Staubli VAL3: Cercle10.pjx

--- Cercle10.pjx ---
Parameters version=s7.3.1 stackSize=5000 millimeterUnit=true
Program file=start.pgx
Program file=stop.pgx
Data file=Cercle10.dtx

--- Cercle10.dtx ---
public frame fReference = {x=1500, y=200, z=-689.53, rz=90, fatherId=world[0]}
public jointRx jPark = {j3=90, j5=90}
public jointRx jJoint = {j1=-0.42016, j2=47.67737, j3=89.12207, j5=43.20056, j6=178.21616}
public mdesc mNomSpeed = {blend=off}
public mdesc mSpeed[30]
  [0] = {tmax=30, rmax=100, leave=0.1, reach=0.1, blend=cartesian}
  [1] = {tmax=30, rmax=100, leave=0.1, reach=0.1, blend=cartesian}
  [2] = {tmax=30, rmax=100, leave=0.1, reach=0.1, blend=cartesian}
  [3] = {tmax=30, rmax=100, leave=0.1, reach=0.1, blend=cartesian}
  [4] = {tmax=30, rmax=100, leave=0.1, reach=0.1, blend=cartesian}
  [5] = {tmax=30, rmax=100, leave=0.1, reach=0.1, blend=cartesian}
  [6] = {tmax=30, rmax=100, leave=0.1, reach=0.1, blend=cartesian}
  [7] = {tmax=30, rmax=100, leave=0.1, reach=0.1, blend=cartesian}
  [8] = {tmax=30, rmax=100, leave=0.1, reach=0.1, blend=cartesian}
  [9] = {tmax=30, rmax=100, leave=0.1, reach=0.1, blend=cartesian}
  [10] = {tmax=30, rmax=100, leave=0.1, reach=0.1, blend=cartesian}
  [11] = {tmax=30, rmax=100, leave=0.1, reach=0.1, blend=cartesian}
  [12] = {tmax=30, rmax=100, leave=0.1, reach=0.1, blend=cartesian}
  [13] = {tmax=30, rmax=100, leave=0.1, reach=0.1, blend=cartesian}
  [14] = {tmax=30, rmax=100, leave=0.1, reach=0.1, blend=cartesian}
  [15] = {tmax=30, rmax=100, leave=0.1, reach=0.1, blend=cartesian}
  [16] = {tmax=30, rmax=100, leave=0.1, reach=0.1, blend=cartesian}
  [17] = {tmax=30, rmax=100, leave=0.1, reach=0.1, blend=cartesian}
  [18] = {tmax=30, rmax=100, leave=0.1, reach=0.1, blend=cartesian}
  [19] = {tmax=30, rmax=100, leave=0.1, reach=0.1, blend=cartesian}
  [20] = {tmax=30, rmax=100, leave=0.1, reach=0.1, blend=cartesian}
  [21] = {tmax=30, rmax=100, leave=0.1, reach=0.1, blend=cartesian}
  [22] = {tmax=30, rmax=100, leave=0.1, reach=0.1, blend=cartesian}
  [23] = {tmax=30, rmax=100, leave=0.1, reach=0.1, blend=cartesian}
  [24] = {tmax=30, rmax=100, leave=0.1, reach=0.1, blend=cartesian}
  [25] = {tmax=30, rmax=100, leave=0.1, reach=0.1, blend=cartesian}
  [26] = {tmax=30, rmax=100, leave=0.1, reach=0.1, blend=cartesian}
  [27] = {tmax=30, rmax=100, leave=0.1, reach=0.1, blend=cartesian}
  [28] = {tmax=30, rmax=100, leave=0.1, reach=0.1, blend=cartesian}
  [29] = {tmax=30, rmax=100, leave=0.1, reach=0.1, blend=cartesian}
public num nTraj
num nTimeStop
num nTimeStart
num nMode
num nEtat
public pointRx pPoint[1370]
  [0] = {x=-211, z=100, rx=-180, rz=88.636, shoulder=lefty, elbow=epositive, wrist=wpositive, fatherId=fReference[0]}
  [1] = {x=-211, rx=-180, rz=88.636, shoulder=lefty, elbow=epositive, wrist=wpositive, fatherId=fReference[0]}
  [2] = {x=-211, rx=-180, rz=88.636, shoulder=lefty, elbow=epositive, wrist=wpositive, fatherId=fReference[0]}
  [3] = {x=-210.761, y=-10.04, rx=-180, rz=85.909, shoulder=lefty, elbow=epositive, wrist=wpositive, fatherId=fReference[0]}
  [4] = {x=-210.045, y=-20.057, rx=-180, rz=83.182, shoulder=lefty, elbow=epositive, wrist=wpositive, fatherId=fReference[0]}
  [5] = {x=-208.852, y=-30.028, rx=-180, rz=80.455, shoulder=lefty, elbow=epositive, wrist=wpositive, fatherId=fReference[0]}
  [6] = {x=-207.187, y=-39.932, rx=-180, rz=77.727, shoulder=lefty, elbow=epositive, wrist=wpositive, fatherId=fReference[0]}
  [7] = {x=-205.052, y=-49.745, rx=-180, rz=75, shoulder=lefty, elbow=epositive, wrist=wpositive, fatherId=fReference[0]}
  [8] = {x=-202.453, y=-59.446, rx=-180, rz=72.273, shoulder=lefty, elbow=epositive, wrist=wpositive, fatherId=fReference[0]}
  [9] = {x=-199.395, y=-69.011, rx=-180, rz=69.545, shoulder=lefty, elbow=epositive, wrist=wpositive, fatherId=fReference[0]}
  [10] = {x=-195.886, y=-78.421, rx=-180, rz=66.818, shoulder=lefty, elbow=epositive, wrist=wpositive, fatherId=fReference[0]}
  [11] = {x=-191.932, y=-87.653, rx=-180, rz=64.091, shoulder=lefty, elbow=epositive, wrist=wpositive, fatherId=fReference[0]}
  [12] = {x=-187.544, y=-96.686, rx=-180, rz=61.364, shoulder=lefty, elbow=epositive, wrist=wpositive, fatherId=fReference[0]}
  [13] = {x=-182.731, y=-105.5, rx=180, rz=58.636, shoulder=lefty, elbow=epositive, wrist=wpositive, fatherId=fReference[0]}
  [14] = {x=-177.505, y=-114.075, rx=-180, rz=55.909, shoulder=lefty, elbow=epositive, wrist=wpositive, fatherId=fReference[0]}
  [15] = {x=-171.876, y=-122.392, rx=-180, rz=53.182, shoulder=lefty, elbow=epositive, wrist=wpositive, fatherId=fReference[0]}
  [16] = {x=-165.857, y=-130.432, rx=-180, rz=50.455, shoulder=lefty, elbow=epositive, wrist=wpositive, fatherId=fReference[0]}
  [17] = {x=-159.463, y=-138.176, rx=-180, rz=47.727, shoulder=lefty, elbow=epositive, wrist=wpositive, fatherId=fReference[0]}
  [18] = {x=-152.708, y=-145.607, rx=-180, rz=45, shoulder=lefty, elbow=epositive, wrist=wpositive, fatherId=fReference[0]}
  [19] = {x=-145.607, y=-152.708, rx=-180, rz=42.273, shoulder=lefty, elbow=epositive, wrist=wpositive, fatherId=fReference[0]}
  [20] = {x=-138.176, y=-159.463, rx=-180, rz=39.545, shoulder=lefty, elbow=epositive, wrist=wpositive, fatherId=fReference[0]}
  [21] = {x=-130.432, y=-165.857, rx=180, rz=36.818, shoulder=lefty, elbow=epositive, wrist=wpositive, fatherId=fReference[0]}
  [22] = {x=-122.392, y=-171.876, rx=180, rz=34.091, shoulder=lefty, elbow=epositive, wrist=wpositive, fatherId=fReference[0]}
  [23] = {x=-114.075, y=-177.505, rx=-180, rz=31.364, shoulder=lefty, elbow=epositive, wrist=wpositive, fatherId=fReference[0]}
  [24] = {x=-105.5, y=-182.731, rx=-180, rz=28.636, shoulder=lefty, elbow=epositive, wrist=wpositive, fatherId=fReference[0]}
  [25] = {x=-96.686, y=-187.544, rx=-180, rz=25.909, shoulder=lefty, elbow=epositive, wrist=wpositive, fatherId=fReference[0]}
  [26] = {x=-87.653, y=-191.932, rx=-180, rz=23.182, shoulder=lefty, elbow=epositive, wrist=wpositive, fatherId=fReference[0]}
  [27] = {x=-78.421, y=-195.886, rx=-180, rz=20.455, shoulder=lefty, elbow=epositive, wrist=wpositive, fatherId=fReference[0]}
  [28] = {x=-69.011, y=-199.395, rx=-180, rz=17.727, shoulder=lefty, elbow=epositive, wrist=wpositive, fatherId=fReference[0]}
  [29] = {x=-59.446, y=-202.453, rx=180, rz=15, shoulder=lefty, elbow=epositive, wrist=wpositive, fatherId=fReference[0]}
  [30] = {x=-49.745, y=-205.052, rx=180, rz=12.273, shoulder=lefty, elbow=epositive, wrist=wpositive, fatherId=fReference[0]}
  [31] = {x=-39.932, y=-207.187, rx=180, rz=9.545, shoulder=lefty, elbow=epositive, wrist=wpositive, fatherId=fReference[0]}
  [32] = {x=-30.028, y=-208.852, rx=-180, rz=6.818, shoulder=lefty, elbow=epositive, wrist=wpositive, fatherId=fReference[0]}
  [33] = {x=-20.057, y=-210.045, rx=-180, rz=4.091, shoulder=lefty, elbow=epositive, wrist=wpositive, fatherId=fReference[0]}
  [34] = {x=-10.04, y=-210.761, rx=180, rz=1.364, shoulder=lefty, elbow=epositive, wrist=wpositive, fatherId=fReference[0]}
  [35] = {y=-211, rx=180, rz=-1.364, shoulder=lefty, elbow=epositive, wrist=wpositive, fatherId=fReference[0]}
  [36] = {x=10.04, y=-210.761, rx=180, rz=-4.091, shoulder=lefty, elbow=epositive, wrist=wpositive, fatherId=fReference[0]}
  [37] = {x=20.057, y=-210.045, rx=-180, rz=-6.818, shoulder=lefty, elbow=epositive, wrist=wpositive, fatherId=fReference[0]}
  [38] = {x=30.028, y=-208.852, rx=180, rz=-9.545, shoulder=lefty, elbow=epositive, wrist=wpositive, fatherId=fReference[0]}
  [39] = {x=39.932, y=-207.187, rx=180, rz=-12.273, shoulder=lefty, elbow=epositive, wrist=wpositive, fatherId=fReference[0]}
  [40] = {x=49.745, y=-205.052, rx=-180, rz=-15, shoulder=lefty, elbow=epositive, wrist=wpositive, fatherId=fReference[0]}
  [41] = {x=59.446, y=-202.453, rx=-180, rz=-17.727, shoulder=lefty, elbow=epositive, wrist=wpositive, fatherId=fReference[0]}
  [42] = {x=69.011, y=-199.395, rx=180, rz=-20.455, shoulder=lefty, elbow=epositive, wrist=wpositive, fatherId=fReference[0]}
  [43] = {x=78.421, y=-195.886, rx=-180, rz=-23.182, shoulder=lefty, elbow=epositive, wrist=wpositive, fatherId=fReference[0]}
  [44] = {x=87.653, y=-191.932, rx=-180, rz=-25.909, shoulder=lefty, elbow=epositive, wrist=wpositive, fatherId=fReference[0]}
  [45] = {x=96.686, y=-187.544, rx=180, rz=-28.636, shoulder=lefty, elbow=epositive, wrist=wpositive, fatherId=fReference[0]}
  [46] = {x=105.5, y=-182.731, rx=-180, rz=-31.364, shoulder=lefty, elbow=epositive, wrist=wpositive, fatherId=fReference[0]}
  [47] = {x=114.075, y=-177.505, rx=180, rz=-34.091, shoulder=lefty, elbow=epositive, wrist=wpositive, fatherId=fReference[0]}
  [48] = {x=122.392, y=-171.876, rx=180, rz=-36.818, shoulder=lefty, elbow=epositive, wrist=wpositive, fatherId=fReference[0]}
  [49] = {x=130.432, y=-165.857, rx=180, rz=-39.545, shoulder=lefty, elbow=epositive, wrist=wpositive, fatherId=fReference[0]}
  [50] = {x=138.176, y=-159.463, rx=180, rz=-42.273, shoulder=lefty, elbow=epositive, wrist=wpositive, fatherId=fReference[0]}
  [51] = {x=145.607, y=-152.708, rx=180, rz=-45, shoulder=lefty, elbow=epositive, wrist=wpositive, fatherId=fReference[0]}
  [52] = {x=152.708, y=-145.607, rx=-180, rz=-47.727, shoulder=lefty, elbow=epositive, wrist=wpositive, fatherId=fReference[0]}
  [53] = {x=159.463, y=-138.176, rx=-180, rz=-50.455, shoulder=lefty, elbow=epositive, wrist=wpositive, fatherId=fReference[0]}
  [54] = {x=165.857, y=-130.432, rx=180, rz=-53.182, shoulder=lefty, elbow=epositive, wrist=wpositive, fatherId=fReference[0]}
  [55] = {x=171.876, y=-122.392, rx=-180, rz=-55.909, shoulder=lefty, elbow=epositive, wrist=wpositive, fatherId=fReference[0]}
  [56] = {x=177.505, y=-114.075, rx=180, rz=-58.636, shoulder=lefty, elbow=epositive, wrist=wpositive, fatherId=fReference[0]}
  [57] = {x=182.731, y=-105.5, rx=-180, rz=-61.364, shoulder=lefty, elbow=epositive, wrist=wpositive, fatherId=fReference[0]}
  [58] = {x=187.544, y=-96.686, rx=180, rz=-64.091, shoulder=lefty, elbow=epositive, wrist=wpositive, fatherId=fReference[0]}
  [59] = {x=191.932, y=-87.653, rx=180, rz=-66.818, shoulder=lefty, elbow=epositive, wrist=wpositive, fatherId=fReference[0]}
  [60] = {x=195.886, y=-78.421, rx=180, rz=-69.545, shoulder=lefty, elbow=epositive, wrist=wpositive, fatherId=fReference[0]}
  [61] = {x=199.395, y=-69.011, rx=180, rz=-72.273, shoulder=lefty, elbow=epositive, wrist=wpositive, fatherId=fReference[0]}
  [62] = {x=202.453, y=-59.446, rx=180, rz=-75, shoulder=lefty, elbow=epositive, wrist=wpositive, fatherId=fReference[0]}
  [63] = {x=205.052, y=-49.745, rx=180, rz=-77.727, shoulder=lefty, elbow=epositive, wrist=wpositive, fatherId=fReference[0]}
  [64] = {x=207.187, y=-39.932, rx=180, rz=-80.455, shoulder=lefty, elbow=epositive, wrist=wpositive, fatherId=fReference[0]}
  [65] = {x=208.852, y=-30.028, rx=180, rz=-83.182, shoulder=lefty, elbow=epositive, wrist=wpositive, fatherId=fReference[0]}
  [66] = {x=210.045, y=-20.057, rx=180, rz=-85.909, shoulder=lefty, elbow=epositive, wrist=wpositive, fatherId=fReference[0]}
  [67] = {x=210.761, y=-10.04, rx=180, rz=-88.636, shoulder=lefty, elbow=epositive, wrist=wpositive, fatherId=fReference[0]}
  [68] = {x=211, rx=-180, rz=-91.364, shoulder=lefty, elbow=epositive, wrist=wpositive, fatherId=fReference[0]}
  [69] = {x=210.761, y=10.04, rx=-180, rz=-94.091, shoulder=lefty, elbow=epositive, wrist=wpositive, fatherId=fReference[0]}
  [70] = {x=210.045, y=20.057, rx=-180, rz=-96.818, shoulder=lefty, elbow=epositive, wrist=wpositive, fatherId=fReference[0]}
  [71] = {x=208.852, y=30.028, rx=-180, rz=-99.545, shoulder=lefty, elbow=epositive, wrist=wpositive, fatherId=fReference[0]}
  [72] = {x=207.187, y=39.932, rx=-180, rz=-102.273, shoulder=lefty, elbow=epositive, wrist=wpositive, fatherId=fReference[0]}
  [73] = {x=205.052, y=49.745, rx=-180, rz=-105, shoulder=lefty, elbow=epositive, wrist=wpositive, fatherId=fReference[0]}
  [74] = {x=202.453, y=59.446, rx=-180, rz=-107.727, shoulder=lefty, elbow=epositive, wrist=wpositive, fatherId=fReference[0]}
  [75] = {x=199.395, y=69.011, rx=-180, rz=-110.455, shoulder=lefty, elbow=epositive, wrist=wpositive, fatherId=fReference[0]}
  [76] = {x=195.886, y=78.421, rx=-180, rz=-113.182, shoulder=lefty, elbow=epositive, wrist=wpositive, fatherId=fReference[0]}
  [77] = {x=191.932, y=87.653, rx=-180, rz=-115.909, shoulder=lefty, elbow=epositive, wrist=wpositive, fatherId=fReference[0]}
  [78] = {x=187.544, y=96.686, rx=-180, rz=-118.636, shoulder=lefty, elbow=epositive, wrist=wpositive, fatherId=fReference[0]}
  [79] = {x=182.731, y=105.5, rx=-180, rz=-121.364, shoulder=lefty, elbow=epositive, wrist=wpositive, fatherId=fReference[0]}
  [80] = {x=177.505, y=114.075, rx=-180, rz=-124.091, shoulder=lefty, elbow=epositive, wrist=wpositive, fatherId=fReference[0]}
  [81] = {x=171.876, y=122.392, rx=-180, rz=-126.818, shoulder=lefty, elbow=epositive, wrist=wpositive, fatherId=fReference[0]}
  [82] = {x=165.857, y=130.432, rx=-180, rz=-129.545, shoulder=lefty, elbow=epositive, wrist=wpositive, fatherId=fReference[0]}
  [83] = {x=159.463, y=138.176, rx=-180, rz=-132.273, shoulder=lefty, elbow=epositive, wrist=wpositive, fatherId=fReference[0]}
  [84] = {x=152.708, y=145.607, rx=-180, rz=-135, shoulder=lefty, elbow=epositive, wrist=wpositive, fatherId=fReference[0]}
  [85] = {x=145.607, y=152.708, rx=-180, rz=-137.727, shoulder=lefty, elbow=epositive, wrist=wpositive, fatherId=fReference[0]}
  [86] = {x=138.176, y=159.463, rx=-180, rz=-140.455, shoulder=lefty, elbow=epositive, wrist=wpositive, fatherId=fReference[0]}
  [87] = {x=130.432, y=165.857, rx=180, rz=-143.182, shoulder=lefty, elbow=epositive, wrist=wpositive, fatherId=fReference[0]}
  [88] = {x=122.392, y=171.876, rx=-180, rz=-145.909, shoulder=lefty, elbow=epositive, wrist=wpositive, fatherId=fReference[0]}
  [89] = {x=114.075, y=177.505, rx=-180, rz=-148.636, shoulder=lefty, elbow=epositive, wrist=wpositive, fatherId=fReference[0]}
  [90] = {x=105.5, y=182.731, rx=-180, rz=-151.364, shoulder=lefty, elbow=epositive, wrist=wpositive, fatherId=fReference[0]}
  [91] = {x=96.686, y=187.544, rx=-180, rz=-154.091, shoulder=lefty, elbow=epositive, wrist=wpositive, fatherId=fReference[0]}
  [92] = {x=87.653, y=191.932, rx=180, rz=-156.818, shoulder=lefty, elbow=epositive, wrist=wpositive, fatherId=fReference[0]}
  [93] = {x=78.421, y=195.886, rx=-180, rz=-159.545, shoulder=lefty, elbow=epositive, wrist=wpositive, fatherId=fReference[0]}
  [94] = {x=69.011, y=199.395, rx=180, rz=-162.273, shoulder=lefty, elbow=epositive, wrist=wpositive, fatherId=fReference[0]}
  [95] = {x=59.446, y=202.453, rx=-180, rz=-165, shoulder=lefty, elbow=epositive, wrist=wpositive, fatherId=fReference[0]}
  [96] = {x=49.745, y=205.052, rx=180, rz=-167.727, shoulder=lefty, elbow=epositive, wrist=wpositive, fatherId=fReference[0]}
  [97] = {x=39.932, y=207.187, rx=-180, rz=-170.455, shoulder=lefty, elbow=epositive, wrist=wpositive, fatherId=fReference[0]}
  [98] = {x=30.028, y=208.852, rx=-180, rz=-173.182, shoulder=lefty, elbow=epositive, wrist=wpositive, fatherId=fReference[0]}
  [99] = {x=20.057, y=210.045, rx=-180, rz=-175.909, shoulder=lefty, elbow=epositive, wrist=wpositive, fatherId=fReference[0]}
  [100] = {x=10.04, y=210.761, rx=-180, rz=-178.636, shoulder=lefty, elbow=epositive, wrist=wpositive, fatherId=fReference[0]}
  [101] = {y=211, rx=180, rz=178.636, shoulder=lefty, elbow=epositive, wrist=wpositive, fatherId=fReference[0]}
  [102] = {x=-10.04, y=210.761, rx=180, rz=175.909, shoulder=lefty, elbow=epositive, wrist=wpositive, fatherId=fReference[0]}
  [103] = {x=-20.057, y=210.045, rx=180, rz=173.182, shoulder=lefty, elbow=epositive, wrist=wpositive, fatherId=fReference[0]}
  [104] = {x=-30.028, y=208.852, rx=180, rz=170.455, shoulder=lefty, elbow=epositive, wrist=wpositive, fatherId=fReference[0]}
  [105] = {x=-39.932, y=207.187, rx=-180, rz=167.727, shoulder=lefty, elbow=epositive, wrist=wpositive, fatherId=fReference[0]}
  [106] = {x=-49.745, y=205.052, rx=-180, rz=165, shoulder=lefty, elbow=epositive, wrist=wpositive, fatherId=fReference[0]}
  [107] = {x=-59.446, y=202.453, rx=-180, rz=162.273, shoulder=lefty, elbow=epositive, wrist=wpositive, fatherId=fReference[0]}
  [108] = {x=-69.011, y=199.395, rx=-180, rz=159.545, shoulder=lefty, elbow=epositive, wrist=wpositive, fatherId=fReference[0]}
  [109] = {x=-78.421, y=195.886, rx=180, rz=156.818, shoulder=lefty, elbow=epositive, wrist=wpositive, fatherId=fReference[0]}
  [110] = {x=-87.653, y=191.932, rx=-180, rz=154.091, shoulder=lefty, elbow=epositive, wrist=wpositive, fatherId=fReference[0]}
  [111] = {x=-96.686, y=187.544, rx=180, rz=151.364, shoulder=lefty, elbow=epositive, wrist=wpositive, fatherId=fReference[0]}
  [112] = {x=-105.5, y=182.731, rx=-180, rz=148.636, shoulder=lefty, elbow=epositive, wrist=wpositive, fatherId=fReference[0]}
  [113] = {x=-114.075, y=177.505, rx=180, rz=145.909, shoulder=lefty, elbow=epositive, wrist=wpositive, fatherId=fReference[0]}
  [114] = {x=-122.392, y=171.876, rx=180, rz=143.182, shoulder=lefty, elbow=epositive, wrist=wpositive, fatherId=fReference[0]}
  [115] = {x=-130.432, y=165.857, rx=180, rz=140.455, shoulder=lefty, elbow=epositive, wrist=wpositive, fatherId=fReference[0]}
  [116] = {x=-138.176, y=159.463, rx=-180, rz=137.727, shoulder=lefty, elbow=epositive, wrist=wpositive, fatherId=fReference[0]}
  [117] = {x=-145.607, y=152.708, rx=180, rz=135, shoulder=lefty, elbow=epositive, wrist=wpositive, fatherId=fReference[0]}
  [118] = {x=-152.708, y=145.607, rx=180, rz=132.273, shoulder=lefty, elbow=epositive, wrist=wpositive, fatherId=fReference[0]}
  [119] = {x=-159.463, y=138.176, rx=180, rz=129.545, shoulder=lefty, elbow=epositive, wrist=wpositive, fatherId=fReference[0]}
  [120] = {x=-165.857, y=130.432, rx=180, rz=126.818, shoulder=lefty, elbow=epositive, wrist=wpositive, fatherId=fReference[0]}
  [121] = {x=-171.876, y=122.392, rx=180, rz=124.091, shoulder=lefty, elbow=epositive, wrist=wpositive, fatherId=fReference[0]}
  [122] = {x=-177.505, y=114.075, rx=180, rz=121.364, shoulder=lefty, elbow=epositive, wrist=wpositive, fatherId=fReference[0]}
  [123] = {x=-182.731, y=105.5, rx=180, rz=118.636, shoulder=lefty, elbow=epositive, wrist=wpositive, fatherId=fReference[0]}
  [124] = {x=-187.544, y=96.686, rx=180, rz=115.909, shoulder=lefty, elbow=epositive, wrist=wpositive, fatherId=fReference[0]}
  [125] = {x=-191.932, y=87.653, rx=180, rz=113.182, shoulder=lefty, elbow=epositive, wrist=wpositive, fatherId=fReference[0]}
  [126] = {x=-195.886, y=78.421, rx=180, rz=110.455, shoulder=lefty, elbow=epositive, wrist=wpositive, fatherId=fReference[0]}
  [127] = {x=-199.395, y=69.011, rx=180, rz=107.727, shoulder=lefty, elbow=epositive, wrist=wpositive, fatherId=fReference[0]}
  [128] = {x=-202.453, y=59.446, rx=180, rz=105, shoulder=lefty, elbow=epositive, wrist=wpositive, fatherId=fReference[0]}
  [129] = {x=-205.052, y=49.745, rx=180, rz=102.273, shoulder=lefty, elbow=epositive, wrist=wpositive, fatherId=fReference[0]}
  [130] = {x=-207.187, y=39.932, rx=180, rz=99.545, shoulder=lefty, elbow=epositive, wrist=wpositive, fatherId=fReference[0]}
  [131] = {x=-208.852, y=30.028, rx=180, rz=96.818, shoulder=lefty, elbow=epositive, wrist=wpositive, fatherId=fReference[0]}
  [132] = {x=-210.045, y=20.057, rx=180, rz=94.091, shoulder=lefty, elbow=epositive, wrist=wpositive, fatherId=fReference[0]}
  [133] = {x=-210.761, y=10.04, rx=180, rz=91.364, shoulder=lefty, elbow=epositive, wrist=wpositive, fatherId=fReference[0]}
  [134] = {x=-211, rx=180, rz=91.364, shoulder=lefty, elbow=epositive, wrist=wpositive, fatherId=fReference[0]}
  [135] = {x=-211, rx=180, rz=91.364, shoulder=lefty, elbow=epositive, wrist=wpositive, fatherId=fReference[0]}
  [136] = {x=-211, z=100, rx=180, rz=91.364, shoulder=lefty, elbow=epositive, wrist=wpositive, fatherId=fReference[0]}
  [137] = {x=-211, z=122, rx=180, rz=91.364, shoulder=lefty, elbow=epositive, wrist=wpositive, fatherId=fReference[0]}
  [138] = {x=-211, z=22, rx=180, rz=91.364, shoulder=lefty, elbow=epositive, wrist=wpositive, fatherId=fReference[0]}
  [139] = {x=-211, z=22, rx=180, rz=91.364, shoulder=lefty, elbow=epositive, wrist=wpositive, fatherId=fReference[0]}
  [140] = {x=-210.761, y=10.04, z=22, rx=180, rz=94.091, shoulder=lefty, elbow=epositive, wrist=wpositive, fatherId=fReference[0]}
  [141] = {x=-210.045, y=20.057, z=22, rx=180, rz=96.818, shoulder=lefty, elbow=epositive, wrist=wpositive, fatherId=fReference[0]}
  [142] = {x=-208.852, y=30.028, z=22, rx=180, rz=99.545, shoulder=lefty, elbow=epositive, wrist=wpositive, fatherId=fReference[0]}
  [143] = {x=-207.187, y=39.932, z=22, rx=180, rz=102.273, shoulder=lefty, elbow=epositive, wrist=wpositive, fatherId=fReference[0]}
  [144] = {x=-205.052, y=49.745, z=22, rx=180, rz=105, shoulder=lefty, elbow=epositive, wrist=wpositive, fatherId=fReference[0]}
  [145] = {x=-202.453, y=59.446, z=22, rx=180, rz=107.727, shoulder=lefty, elbow=epositive, wrist=wpositive, fatherId=fReference[0]}
  [146] = {x=-199.395, y=69.011, z=22, rx=180, rz=110.455, shoulder=lefty, elbow=epositive, wrist=wpositive, fatherId=fReference[0]}
  [147] = {x=-195.886, y=78.421, z=22, rx=-180, rz=113.182, shoulder=lefty, elbow=epositive, wrist=wpositive, fatherId=fReference[0]}
  [148] = {x=-191.932, y=87.653, z=22, rx=180, rz=115.909, shoulder=lefty, elbow=epositive, wrist=wpositive, fatherId=fReference[0]}
  [149] = {x=-187.544, y=96.686, z=22, rx=180, rz=118.636, shoulder=lefty, elbow=epositive, wrist=wpositive, fatherId=fReference[0]}
  [150] = {x=-182.731, y=105.5, z=22, rx=180, rz=121.364, shoulder=lefty, elbow=epositive, wrist=wpositive, fatherId=fReference[0]}
  [151] = {x=-177.505, y=114.075, z=22, rx=180, rz=124.091, shoulder=lefty, elbow=epositive, wrist=wpositive, fatherId=fReference[0]}
  [152] = {x=-171.876, y=122.392, z=22, rx=180, rz=126.818, shoulder=lefty, elbow=epositive, wrist=wpositive, fatherId=fReference[0]}
  [153] = {x=-165.857, y=130.432, z=22, rx=180, rz=129.545, shoulder=lefty, elbow=epositive, wrist=wpositive, fatherId=fReference[0]}
  [154] = {x=-159.463, y=138.176, z=22, rx=180, rz=132.273, shoulder=lefty, elbow=epositive, wrist=wpositive, fatherId=fReference[0]}
  [155] = {x=-152.708, y=145.607, z=22, rx=180, rz=135, shoulder=lefty, elbow=epositive, wrist=wpositive, fatherId=fReference[0]}
  [156] = {x=-145.607, y=152.708, z=22, rx=180, rz=137.727, shoulder=lefty, elbow=epositive, wrist=wpositive, fatherId=fReference[0]}
  [157] = {x=-138.176, y=159.463, z=22, rx=180, rz=140.455, shoulder=lefty, elbow=epositive, wrist=wpositive, fatherId=fReference[0]}
  [158] = {x=-130.432, y=165.857, z=22, rx=180, rz=143.182, shoulder=lefty, elbow=epositive, wrist=wpositive, fatherId=fReference[0]}
  [159] = {x=-122.392, y=171.876, z=22, rx=-180, rz=145.909, shoulder=lefty, elbow=epositive, wrist=wpositive, fatherId=fReference[0]}
  [160] = {x=-114.075, y=177.505, z=22, rx=180, rz=148.636, shoulder=lefty, elbow=epositive, wrist=wpositive, fatherId=fReference[0]}
  [161] = {x=-105.5, y=182.731, z=22, rx=180, rz=151.364, shoulder=lefty, elbow=epositive, wrist=wpositive, fatherId=fReference[0]}
  [162] = {x=-96.686, y=187.544, z=22, rx=180, rz=154.091, shoulder=lefty, elbow=epositive, wrist=wpositive, fatherId=fReference[0]}
  [163] = {x=-87.653, y=191.932, z=22, rx=-180, rz=156.818, shoulder=lefty, elbow=epositive, wrist=wpositive, fatherId=fReference[0]}
  [164] = {x=-78.421, y=195.886, z=22, rx=180, rz=159.545, shoulder=lefty, elbow=epositive, wrist=wpositive, fatherId=fReference[0]}
  [165] = {x=-69.011, y=199.395, z=22, rx=-180, rz=162.273, shoulder=lefty, elbow=epositive, wrist=wpositive, fatherId=fReference[0]}
  [166] = {x=-59.446, y=202.453, z=22, rx=-180, rz=165, shoulder=lefty, elbow=epositive, wrist=wpositive, fatherId=fReference[0]}
  [167] = {x=-49.745, y=205.052, z=22, rx=180, rz=167.727, shoulder=lefty, elbow=epositive, wrist=wpositive, fatherId=fReference[0]}
  [168] = {x=-39.932, y=207.187, z=22, rx=-180, rz=170.455, shoulder=lefty, elbow=epositive, wrist=wpositive, fatherId=fReference[0]}
  [169] = {x=-30.028, y=208.852, z=22, rx=180, rz=173.182, shoulder=lefty, elbow=epositive, wrist=wpositive, fatherId=fReference[0]}
  [170] = {x=-20.057, y=210.045, z=22, rx=-180, rz=175.909, shoulder=lefty, elbow=epositive, wrist=wpositive, fatherId=fReference[0]}
  [171] = {x=-10.04, y=210.761, z=22, rx=-180, rz=178.636, shoulder=lefty, elbow=epositive, wrist=wpositive, fatherId=fReference[0]}
  [172] = {y=211, z=22, rx=-180, rz=-178.636, shoulder=lefty, elbow=epositive, wrist=wpositive, fatherId=fReference[0]}
  [173] = {x=10.04, y=210.761, z=22, rx=180, rz=-175.909, shoulder=lefty, elbow=epositive, wrist=wpositive, fatherId=fReference[0]}
  [174] = {x=20.057, y=210.045, z=22, rx=-180, rz=-173.182, shoulder=lefty, elbow=epositive, wrist=wpositive, fatherId=fReference[0]}
  [175] = {x=30.028, y=208.852, z=22, rx=180, rz=-170.455, shoulder=lefty, elbow=epositive, wrist=wpositive, fatherId=fReference[0]}
  [176] = {x=39.932, y=207.187, z=22, rx=180, rz=-167.727, shoulder=lefty, elbow=epositive, wrist=wpositive, fatherId=fReference[0]}
  [177] = {x=49.745, y=205.052, z=22, rx=-180, rz=-165, shoulder=lefty, elbow=epositive, wrist=wpositive, fatherId=fReference[0]}
  [178] = {x=59.446, y=202.453, z=22, rx=-180, rz=-162.273, shoulder=lefty, elbow=epositive, wrist=wpositive, fatherId=fReference[0]}
  [179] = {x=69.011, y=199.395, z=22, rx=-180, rz=-159.545, shoulder=lefty, elbow=epositive, wrist=wpositive, fatherId=fReference[0]}
  [180] = {x=78.421, y=195.886, z=22, rx=180, rz=-156.818, shoulder=lefty, elbow=epositive, wrist=wpositive, fatherId=fReference[0]}
  [181] = {x=87.653, y=191.932, z=22, rx=180, rz=-154.091, shoulder=lefty, elbow=epositive, wrist=wpositive, fatherId=fReference[0]}
  [182] = {x=96.686, y=187.544, z=22, rx=-180, rz=-151.364, shoulder=lefty, elbow=epositive, wrist=wpositive, fatherId=fReference[0]}
  [183] = {x=105.5, y=182.731, z=22, rx=-180, rz=-148.636, shoulder=lefty, elbow=epositive, wrist=wpositive, fatherId=fReference[0]}
  [184] = {x=114.075, y=177.505, z=22, rx=-180, rz=-145.909, shoulder=lefty, elbow=epositive, wrist=wpositive, fatherId=fReference[0]}
  [185] = {x=122.392, y=171.876, z=22, rx=-180, rz=-143.182, shoulder=lefty, elbow=epositive, wrist=wpositive, fatherId=fReference[0]}
  [186] = {x=130.432, y=165.857, z=22, rx=-180, rz=-140.455, shoulder=lefty, elbow=epositive, wrist=wpositive, fatherId=fReference[0]}
  [187] = {x=138.176, y=159.463, z=22, rx=-180, rz=-137.727, shoulder=lefty, elbow=epositive, wrist=wpositive, fatherId=fReference[0]}
  [188] = {x=145.607, y=152.708, z=22, rx=-180, rz=-135, shoulder=lefty, elbow=epositive, wrist=wpositive, fatherId=fReference[0]}
  [189] = {x=152.708, y=145.607, z=22, rx=-180, rz=-132.273, shoulder=lefty, elbow=epositive, wrist=wpositive, fatherId=fReference[0]}
  [190] = {x=159.463, y=138.176, z=22, rx=-180, rz=-129.545, shoulder=lefty, elbow=epositive, wrist=wpositive, fatherId=fReference[0]}
  [191] = {x=165.857, y=130.432, z=22, rx=-180, rz=-126.818, shoulder=lefty, elbow=epositive, wrist=wpositive, fatherId=fReference[0]}
  [192] = {x=171.876, y=122.392, z=22, rx=-180, rz=-124.091, shoulder=lefty, elbow=epositive, wrist=wpositive, fatherId=fReference[0]}
  [193] = {x=177.505, y=114.075, z=22, rx=-180, rz=-121.364, shoulder=lefty, elbow=epositive, wrist=wpositive, fatherId=fReference[0]}
  [194] = {x=182.731, y=105.5, z=22, rx=-180, rz=-118.636, shoulder=lefty, elbow=epositive, wrist=wpositive, fatherId=fReference[0]}
  [195] = {x=187.544, y=96.686, z=22, rx=-180, rz=-115.909, shoulder=lefty, elbow=epositive, wrist=wpositive, fatherId=fReference[0]}
  [196] = {x=191.932, y=87.653, z=22, rx=-180, rz=-113.182, shoulder=lefty, elbow=epositive, wrist=wpositive, fatherId=fReference[0]}
  [197] = {x=195.886, y=78.421, z=22, rx=-180, rz=-110.455, shoulder=lefty, elbow=epositive, wrist=wpositive, fatherId=fReference[0]}
  [198] = {x=199.395, y=69.011, z=22, rx=-180, rz=-107.727, shoulder=lefty, elbow=epositive, wrist=wpositive, fatherId=fReference[0]}
  [199] = {x=202.453, y=59.446, z=22, rx=-180, rz=-105, shoulder=lefty, elbow=epositive, wrist=wpositive, fatherId=fReference[0]}
  [200] = {x=205.052, y=49.745, z=22, rx=-180, rz=-102.273, shoulder=lefty, elbow=epositive, wrist=wpositive, fatherId=fReference[0]}
  [201] = {x=207.187, y=39.932, z=22, rx=-180, rz=-99.545, shoulder=lefty, elbow=epositive, wrist=wpositive, fatherId=fReference[0]}
  [202] = {x=208.852, y=30.028, z=22, rx=-180, rz=-96.818, shoulder=lefty, elbow=epositive, wrist=wpositive, fatherId=fReference[0]}
  [203] = {x=210.045, y=20.057, z=22, rx=-180, rz=-94.091, shoulder=lefty, elbow=epositive, wrist=wpositive, fatherId=fReference[0]}
  [204] = {x=210.761, y=10.04, z=22, rx=-180, rz=-91.364, shoulder=lefty, elbow=epositive, wrist=wpositive, fatherId=fReference[0]}
  [205] = {x=211, z=22, rx=180, rz=-88.636, shoulder=lefty, elbow=epositive, wrist=wpositive, fatherId=fReference[0]}
  [206] = {x=210.761, y=-10.04, z=22, rx=180, rz=-85.909, shoulder=lefty, elbow=epositive, wrist=wpositive, fatherId=fReference[0]}
  [207] = {x=210.045, y=-20.057, z=22, rx=180, rz=-83.182, shoulder=lefty, elbow=epositive, wrist=wpositive, fatherId=fReference[0]}
  [208] = {x=208.852, y=-30.028, z=22, rx=180, rz=-80.455, shoulder=lefty, elbow=epositive, wrist=wpositive, fatherId=fReference[0]}
  [209] = {x=207.187, y=-39.932, z=22, rx=180, rz=-77.727, shoulder=lefty, elbow=epositive, wrist=wpositive, fatherId=fReference[0]}
  [210] = {x=205.052, y=-49.745, z=22, rx=180, rz=-75, shoulder=lefty, elbow=epositive, wrist=wpositive, fatherId=fReference[0]}
  [211] = {x=202.453, y=-59.446, z=22, rx=180, rz=-72.273, shoulder=lefty, elbow=epositive, wrist=wpositive, fatherId=fReference[0]}
  [212] = {x=199.395, y=-69.011, z=22, rx=180, rz=-69.545, shoulder=lefty, elbow=epositive, wrist=wpositive, fatherId=fReference[0]}
  [213] = {x=195.886, y=-78.421, z=22, rx=180, rz=-66.818, shoulder=lefty, elbow=epositive, wrist=wpositive, fatherId=fReference[0]}
  [214] = {x=191.932, y=-87.653, z=22, rx=180, rz=-64.091, shoulder=lefty, elbow=epositive, wrist=wpositive, fatherId=fReference[0]}
  [215] = {x=187.544, y=-96.686, z=22, rx=-180, rz=-61.364, shoulder=lefty, elbow=epositive, wrist=wpositive, fatherId=fReference[0]}
  [216] = {x=182.731, y=-105.5, z=22, rx=-180, rz=-58.636, shoulder=lefty, elbow=epositive, wrist=wpositive, fatherId=fReference[0]}
  [217] = {x=177.505, y=-114.075, z=22, rx=180, rz=-55.909, shoulder=lefty, elbow=epositive, wrist=wpositive, fatherId=fReference[0]}
  [218] = {x=171.876, y=-122.392, z=22, rx=180, rz=-53.182, shoulder=lefty, elbow=epositive, wrist=wpositive, fatherId=fReference[0]}
  [219] = {x=165.857, y=-130.432, z=22, rx=180, rz=-50.455, shoulder=lefty, elbow=epositive, wrist=wpositive, fatherId=fReference[0]}
  [220] = {x=159.463, y=-138.176, z=22, rx=180, rz=-47.727, shoulder=lefty, elbow=epositive, wrist=wpositive, fatherId=fReference[0]}
  [221] = {x=152.708, y=-145.607, z=22, rx=180, rz=-45, shoulder=lefty, elbow=epositive, wrist=wpositive, fatherId=fReference[0]}
  [222] = {x=145.607, y=-152.708, z=22, rx=180, rz=-42.273, shoulder=lefty, elbow=epositive, wrist=wpositive, fatherId=fReference[0]}
  [223] = {x=138.176, y=-159.463, z=22, rx=180, rz=-39.545, shoulder=lefty, elbow=epositive, wrist=wpositive, fatherId=fReference[0]}
  [224] = {x=130.432, y=-165.857, z=22, rx=180, rz=-36.818, shoulder=lefty, elbow=epositive, wrist=wpositive, fatherId=fReference[0]}
  [225] = {x=122.392, y=-171.876, z=22, rx=-180, rz=-34.091, shoulder=lefty, elbow=epositive, wrist=wpositive, fatherId=fReference[0]}
  [226] = {x=114.075, y=-177.505, z=22, rx=180, rz=-31.364, shoulder=lefty, elbow=epositive, wrist=wpositive, fatherId=fReference[0]}
  [227] = {x=105.5, y=-182.731, z=22, rx=180, rz=-28.636, shoulder=lefty, elbow=epositive, wrist=wpositive, fatherId=fReference[0]}
  [228] = {x=96.686, y=-187.544, z=22, rx=-180, rz=-25.909, shoulder=lefty, elbow=epositive, wrist=wpositive, fatherId=fReference[0]}
  [229] = {x=87.653, y=-191.932, z=22, rx=-180, rz=-23.182, shoulder=lefty, elbow=epositive, wrist=wpositive, fatherId=fReference[0]}
  [230] = {x=78.421, y=-195.886, z=22, rx=180, rz=-20.455, shoulder=lefty, elbow=epositive, wrist=wpositive, fatherId=fReference[0]}
  [231] = {x=69.011, y=-199.395, z=22, rx=180, rz=-17.727, shoulder=lefty, elbow=epositive, wrist=wpositive, fatherId=fReference[0]}
  [232] = {x=59.446, y=-202.453, z=22, rx=180, rz=-15, shoulder=lefty, elbow=epositive, wrist=wpositive, fatherId=fReference[0]}
  [233] = {x=49.745, y=-205.052, z=22, rx=180, rz=-12.273, shoulder=lefty, elbow=epositive, wrist=wpositive, fatherId=fReference[0]}
  [234] = {x=39.932, y=-207.187, z=22, rx=-180, rz=-9.545, shoulder=lefty, elbow=epositive, wrist=wpositive, fatherId=fReference[0]}
  [235] = {x=30.028, y=-208.852, z=22, rx=-180, rz=-6.818, shoulder=lefty, elbow=epositive, wrist=wpositive, fatherId=fReference[0]}
  [236] = {x=20.057, y=-210.045, z=22, rx=-180, rz=-4.091, shoulder=lefty, elbow=epositive, wrist=wpositive, fatherId=fReference[0]}
  [237] = {x=10.04, y=-210.761, z=22, rx=-180, rz=-1.364, shoulder=lefty, elbow=epositive, wrist=wpositive, fatherId=fReference[0]}
  [238] = {y=-211, z=22, rx=-180, rz=1.364, shoulder=lefty, elbow=epositive, wrist=wpositive, fatherId=fReference[0]}
  [239] = {x=-10.04, y=-210.761, z=22, rx=-180, rz=4.091, shoulder=lefty, elbow=epositive, wrist=wpositive, fatherId=fReference[0]}
  [240] = {x=-20.057, y=-210.045, z=22, rx=180, rz=6.818, shoulder=lefty, elbow=epositive, wrist=wpositive, fatherId=fReference[0]}
  [241] = {x=-30.028, y=-208.852, z=22, rx=-180, rz=9.545, shoulder=lefty, elbow=epositive, wrist=wpositive, fatherId=fReference[0]}
  [242] = {x=-39.932, y=-207.187, z=22, rx=-180, rz=12.273, shoulder=lefty, elbow=epositive, wrist=wpositive, fatherId=fReference[0]}
  [243] = {x=-49.745, y=-205.052, z=22, rx=180, rz=15, shoulder=lefty, elbow=epositive, wrist=wpositive, fatherId=fReference[0]}
  [244] = {x=-59.446, y=-202.453, z=22, rx=180, rz=17.727, shoulder=lefty, elbow=epositive, wrist=wpositive, fatherId=fReference[0]}
  [245] = {x=-69.011, y=-199.395, z=22, rx=-180, rz=20.455, shoulder=lefty, elbow=epositive, wrist=wpositive, fatherId=fReference[0]}
  [246] = {x=-78.421, y=-195.886, z=22, rx=-180, rz=23.182, shoulder=lefty, elbow=epositive, wrist=wpositive, fatherId=fReference[0]}
  [247] = {x=-87.653, y=-191.932, z=22, rx=-180, rz=25.909, shoulder=lefty, elbow=epositive, wrist=wpositive, fatherId=fReference[0]}
  [248] = {x=-96.686, y=-187.544, z=22, rx=-180, rz=28.636, shoulder=lefty, elbow=epositive, wrist=wpositive, fatherId=fReference[0]}
  [249] = {x=-105.5, y=-182.731, z=22, rx=-180, rz=31.364, shoulder=lefty, elbow=epositive, wrist=wpositive, fatherId=fReference[0]}
  [250] = {x=-114.075, y=-177.505, z=22, rx=-180, rz=34.091, shoulder=lefty, elbow=epositive, wrist=wpositive, fatherId=fReference[0]}
  [251] = {x=-122.392, y=-171.876, z=22, rx=180, rz=36.818, shoulder=lefty, elbow=epositive, wrist=wpositive, fatherId=fReference[0]}
  [252] = {x=-130.432, y=-165.857, z=22, rx=-180, rz=39.545, shoulder=lefty, elbow=epositive, wrist=wpositive, fatherId=fReference[0]}
  [253] = {x=-138.176, y=-159.463, z=22, rx=-180, rz=42.273, shoulder=lefty, elbow=epositive, wrist=wpositive, fatherId=fReference[0]}
  [254] = {x=-145.607, y=-152.708, z=22, rx=-180, rz=45, shoulder=lefty, elbow=epositive, wrist=wpositive, fatherId=fReference[0]}
  [255] = {x=-152.708, y=-145.607, z=22, rx=-180, rz=47.727, shoulder=lefty, elbow=epositive, wrist=wpositive, fatherId=fReference[0]}
  [256] = {x=-159.463, y=-138.176, z=22, rx=-180, rz=50.455, shoulder=lefty, elbow=epositive, wrist=wpositive, fatherId=fReference[0]}
  [257] = {x=-165.857, y=-130.432, z=22, rx=-180, rz=53.182, shoulder=lefty, elbow=epositive, wrist=wpositive, fatherId=fReference[0]}
  [258] = {x=-171.876, y=-122.392, z=22, rx=-180, rz=55.909, shoulder=lefty, elbow=epositive, wrist=wpositive, fatherId=fReference[0]}
  [259] = {x=-177.505, y=-114.075, z=22, rx=-180, rz=58.636, shoulder=lefty, elbow=epositive, wrist=wpositive, fatherId=fReference[0]}
  [260] = {x=-182.731, y=-105.5, z=22, rx=-180, rz=61.364, shoulder=lefty, elbow=epositive, wrist=wpositive, fatherId=fReference[0]}
  [261] = {x=-187.544, y=-96.686, z=22, rx=-180, rz=64.091, shoulder=lefty, elbow=epositive, wrist=wpositive, fatherId=fReference[0]}
  [262] = {x=-191.932, y=-87.653, z=22, rx=-180, rz=66.818, shoulder=lefty, elbow=epositive, wrist=wpositive, fatherId=fReference[0]}
  [263] = {x=-195.886, y=-78.421, z=22, rx=-180, rz=69.545, shoulder=lefty, elbow=epositive, wrist=wpositive, fatherId=fReference[0]}
  [264] = {x=-199.395, y=-69.011, z=22, rx=-180, rz=72.273, shoulder=lefty, elbow=epositive, wrist=wpositive, fatherId=fReference[0]}
  [265] = {x=-202.453, y=-59.446, z=22, rx=-180, rz=75, shoulder=lefty, elbow=epositive, wrist=wpositive, fatherId=fReference[0]}
  [266] = {x=-205.052, y=-49.745, z=22, rx=-180, rz=77.727, shoulder=lefty, elbow=epositive, wrist=wpositive, fatherId=fReference[0]}
  [267] = {x=-207.187, y=-39.932, z=22, rx=-180, rz=80.455, shoulder=lefty, elbow=epositive, wrist=wpositive, fatherId=fReference[0]}
  [268] = {x=-208.852, y=-30.028, z=22, rx=-180, rz=83.182, shoulder=lefty, elbow=epositive, wrist=wpositive, fatherId=fReference[0]}
  [269] = {x=-210.045, y=-20.057, z=22, rx=-180, rz=85.909, shoulder=lefty, elbow=epositive, wrist=wpositive, fatherId=fReference[0]}
  [270] = {x=-210.761, y=-10.04, z=22, rx=-180, rz=88.636, shoulder=lefty, elbow=epositive, wrist=wpositive, fatherId=fReference[0]}
  [271] = {x=-211, z=22, rx=-180, rz=88.636, shoulder=lefty, elbow=epositive, wrist=wpositive, fatherId=fReference[0]}
  [272] = {x=-211, z=22, rx=-180, rz=88.636, shoulder=lefty, elbow=epositive, wrist=wpositive, fatherId=fReference[0]}
  [273] = {x=-211, z=122, rx=-180, rz=88.636, shoulder=lefty, elbow=epositive, wrist=wpositive, fatherId=fReference[0]}
  [274] = {x=-211, z=144, rx=-180, rz=88.636, shoulder=lefty, elbow=epositive, wrist=wpositive, fatherId=fReference[0]}
  [275] = {x=-211, z=44, rx=-180, rz=88.636, shoulder=lefty, elbow=epositive, wrist=wpositive, fatherId=fReference[0]}
  [276] = {x=-211, z=44, rx=-180, rz=88.636, shoulder=lefty, elbow=epositive, wrist=wpositive, fatherId=fReference[0]}
  [277] = {x=-210.761, y=-10.04, z=44, rx=-180, rz=85.909, shoulder=lefty, elbow=epositive, wrist=wpositive, fatherId=fReference[0]}
  [278] = {x=-210.045, y=-20.057, z=44, rx=-180, rz=83.182, shoulder=lefty, elbow=epositive, wrist=wpositive, fatherId=fReference[0]}
  [279] = {x=-208.852, y=-30.028, z=44, rx=-180, rz=80.455, shoulder=lefty, elbow=epositive, wrist=wpositive, fatherId=fReference[0]}
  [280] = {x=-207.187, y=-39.932, z=44, rx=-180, rz=77.727, shoulder=lefty, elbow=epositive, wrist=wpositive, fatherId=fReference[0]}
  [281] = {x=-205.052, y=-49.745, z=44, rx=-180, rz=75, shoulder=lefty, elbow=epositive, wrist=wpositive, fatherId=fReference[0]}
  [282] = {x=-202.453, y=-59.446, z=44, rx=-180, rz=72.273, shoulder=lefty, elbow=epositive, wrist=wpositive, fatherId=fReference[0]}
  [283] = {x=-199.395, y=-69.011, z=44, rx=-180, rz=69.545, shoulder=lefty, elbow=epositive, wrist=wpositive, fatherId=fReference[0]}
  [284] = {x=-195.886, y=-78.421, z=44, rx=-180, rz=66.818, shoulder=lefty, elbow=epositive, wrist=wpositive, fatherId=fReference[0]}
  [285] = {x=-191.932, y=-87.653, z=44, rx=-180, rz=64.091, shoulder=lefty, elbow=epositive, wrist=wpositive, fatherId=fReference[0]}
  [286] = {x=-187.544, y=-96.686, z=44, rx=-180, rz=61.364, shoulder=lefty, elbow=epositive, wrist=wpositive, fatherId=fReference[0]}
  [287] = {x=-182.731, y=-105.5, z=44, rx=-180, rz=58.636, shoulder=lefty, elbow=epositive, wrist=wpositive, fatherId=fReference[0]}
  [288] = {x=-177.505, y=-114.075, z=44, rx=-180, rz=55.909, shoulder=lefty, elbow=epositive, wrist=wpositive, fatherId=fReference[0]}
  [289] = {x=-171.876, y=-122.392, z=44, rx=-180, rz=53.182, shoulder=lefty, elbow=epositive, wrist=wpositive, fatherId=fReference[0]}
  [290] = {x=-165.857, y=-130.432, z=44, rx=-180, rz=50.455, shoulder=lefty, elbow=epositive, wrist=wpositive, fatherId=fReference[0]}
  [291] = {x=-159.463, y=-138.176, z=44, rx=-180, rz=47.727, shoulder=lefty, elbow=epositive, wrist=wpositive, fatherId=fReference[0]}
  [292] = {x=-152.708, y=-145.607, z=44, rx=-180, rz=45, shoulder=lefty, elbow=epositive, wrist=wpositive, fatherId=fReference[0]}
  [293] = {x=-145.607, y=-152.708, z=44, rx=-180, rz=42.273, shoulder=lefty, elbow=epositive, wrist=wpositive, fatherId=fReference[0]}
  [294] = {x=-138.176, y=-159.463, z=44, rx=-180, rz=39.545, shoulder=lefty, elbow=epositive, wrist=wpositive, fatherId=fReference[0]}
  [295] = {x=-130.432, y=-165.857, z=44, rx=-180, rz=36.818, shoulder=lefty, elbow=epositive, wrist=wpositive, fatherId=fReference[0]}
  [296] = {x=-122.392, y=-171.876, z=44, rx=-180, rz=34.091, shoulder=lefty, elbow=epositive, wrist=wpositive, fatherId=fReference[0]}
  [297] = {x=-114.075, y=-177.505, z=44, rx=-180, rz=31.364, shoulder=lefty, elbow=epositive, wrist=wpositive, fatherId=fReference[0]}
  [298] = {x=-105.5, y=-182.731, z=44, rx=-180, rz=28.636, shoulder=lefty, elbow=epositive, wrist=wpositive, fatherId=fReference[0]}
  [299] = {x=-96.686, y=-187.544, z=44, rx=-180, rz=25.909, shoulder=lefty, elbow=epositive, wrist=wpositive, fatherId=fReference[0]}
  [300] = {x=-87.653, y=-191.932, z=44, rx=180, rz=23.182, shoulder=lefty, elbow=epositive, wrist=wpositive, fatherId=fReference[0]}
  [301] = {x=-78.421, y=-195.886, z=44, rx=180, rz=20.455, shoulder=lefty, elbow=epositive, wrist=wpositive, fatherId=fReference[0]}
  [302] = {x=-69.011, y=-199.395, z=44, rx=-180, rz=17.727, shoulder=lefty, elbow=epositive, wrist=wpositive, fatherId=fReference[0]}
  [303] = {x=-59.446, y=-202.453, z=44, rx=-180, rz=15, shoulder=lefty, elbow=epositive, wrist=wpositive, fatherId=fReference[0]}
  [304] = {x=-49.745, y=-205.052, z=44, rx=-180, rz=12.273, shoulder=lefty, elbow=epositive, wrist=wpositive, fatherId=fReference[0]}
  [305] = {x=-39.932, y=-207.187, z=44, rx=-180, rz=9.545, shoulder=lefty, elbow=epositive, wrist=wpositive, fatherId=fReference[0]}
  [306] = {x=-30.028, y=-208.852, z=44, rx=-180, rz=6.818, shoulder=lefty, elbow=epositive, wrist=wpositive, fatherId=fReference[0]}
  [307] = {x=-20.057, y=-210.045, z=44, rx=180, rz=4.091, shoulder=lefty, elbow=epositive, wrist=wpositive, fatherId=fReference[0]}
  [308] = {x=-10.04, y=-210.761, z=44, rx=-180, rz=1.364, shoulder=lefty, elbow=epositive, wrist=wpositive, fatherId=fReference[0]}
  [309] = {y=-211, z=44, rx=180, rz=-1.364, shoulder=lefty, elbow=epositive, wrist=wpositive, fatherId=fReference[0]}
  [310] = {x=10.04, y=-210.761, z=44, rx=-180, rz=-4.091, shoulder=lefty, elbow=epositive, wrist=wpositive, fatherId=fReference[0]}
  [311] = {x=20.057, y=-210.045, z=44, rx=180, rz=-6.818, shoulder=lefty, elbow=epositive, wrist=wpositive, fatherId=fReference[0]}
  [312] = {x=30.028, y=-208.852, z=44, rx=180, rz=-9.545, shoulder=lefty, elbow=epositive, wrist=wpositive, fatherId=fReference[0]}
  [313] = {x=39.932, y=-207.187, z=44, rx=-180, rz=-12.273, shoulder=lefty, elbow=epositive, wrist=wpositive, fatherId=fReference[0]}
  [314] = {x=49.745, y=-205.052, z=44, rx=-180, rz=-15, shoulder=lefty, elbow=epositive, wrist=wpositive, fatherId=fReference[0]}
  [315] = {x=59.446, y=-202.453, z=44, rx=180, rz=-17.727, shoulder=lefty, elbow=epositive, wrist=wpositive, fatherId=fReference[0]}
  [316] = {x=69.011, y=-199.395, z=44, rx=180, rz=-20.455, shoulder=lefty, elbow=epositive, wrist=wpositive, fatherId=fReference[0]}
  [317] = {x=78.421, y=-195.886, z=44, rx=180, rz=-23.182, shoulder=lefty, elbow=epositive, wrist=wpositive, fatherId=fReference[0]}
  [318] = {x=87.653, y=-191.932, z=44, rx=180, rz=-25.909, shoulder=lefty, elbow=epositive, wrist=wpositive, fatherId=fReference[0]}
  [319] = {x=96.686, y=-187.544, z=44, rx=-180, rz=-28.636, shoulder=lefty, elbow=epositive, wrist=wpositive, fatherId=fReference[0]}
  [320] = {x=105.5, y=-182.731, z=44, rx=180, rz=-31.364, shoulder=lefty, elbow=epositive, wrist=wpositive, fatherId=fReference[0]}
  [321] = {x=114.075, y=-177.505, z=44, rx=180, rz=-34.091, shoulder=lefty, elbow=epositive, wrist=wpositive, fatherId=fReference[0]}
  [322] = {x=122.392, y=-171.876, z=44, rx=180, rz=-36.818, shoulder=lefty, elbow=epositive, wrist=wpositive, fatherId=fReference[0]}
  [323] = {x=130.432, y=-165.857, z=44, rx=180, rz=-39.545, shoulder=lefty, elbow=epositive, wrist=wpositive, fatherId=fReference[0]}
  [324] = {x=138.176, y=-159.463, z=44, rx=180, rz=-42.273, shoulder=lefty, elbow=epositive, wrist=wpositive, fatherId=fReference[0]}
  [325] = {x=145.607, y=-152.708, z=44, rx=180, rz=-45, shoulder=lefty, elbow=epositive, wrist=wpositive, fatherId=fReference[0]}
  [326] = {x=152.708, y=-145.607, z=44, rx=180, rz=-47.727, shoulder=lefty, elbow=epositive, wrist=wpositive, fatherId=fReference[0]}
  [327] = {x=159.463, y=-138.176, z=44, rx=180, rz=-50.455, shoulder=lefty, elbow=epositive, wrist=wpositive, fatherId=fReference[0]}
  [328] = {x=165.857, y=-130.432, z=44, rx=-180, rz=-53.182, shoulder=lefty, elbow=epositive, wrist=wpositive, fatherId=fReference[0]}
  [329] = {x=171.876, y=-122.392, z=44, rx=-180, rz=-55.909, shoulder=lefty, elbow=epositive, wrist=wpositive, fatherId=fReference[0]}
  [330] = {x=177.505, y=-114.075, z=44, rx=180, rz=-58.636, shoulder=lefty, elbow=epositive, wrist=wpositive, fatherId=fReference[0]}
  [331] = {x=182.731, y=-105.5, z=44, rx=-180, rz=-61.364, shoulder=lefty, elbow=epositive, wrist=wpositive, fatherId=fReference[0]}
  [332] = {x=187.544, y=-96.686, z=44, rx=-180, rz=-64.091, shoulder=lefty, elbow=epositive, wrist=wpositive, fatherId=fReference[0]}
  [333] = {x=191.932, y=-87.653, z=44, rx=-180, rz=-66.818, shoulder=lefty, elbow=epositive, wrist=wpositive, fatherId=fReference[0]}
  [334] = {x=195.886, y=-78.421, z=44, rx=-180, rz=-69.545, shoulder=lefty, elbow=epositive, wrist=wpositive, fatherId=fReference[0]}
  [335] = {x=199.395, y=-69.011, z=44, rx=180, rz=-72.273, shoulder=lefty, elbow=epositive, wrist=wpositive, fatherId=fReference[0]}
  [336] = {x=202.453, y=-59.446, z=44, rx=180, rz=-75, shoulder=lefty, elbow=epositive, wrist=wpositive, fatherId=fReference[0]}
  [337] = {x=205.052, y=-49.745, z=44, rx=180, rz=-77.727, shoulder=lefty, elbow=epositive, wrist=wpositive, fatherId=fReference[0]}
  [338] = {x=207.187, y=-39.932, z=44, rx=180, rz=-80.455, shoulder=lefty, elbow=epositive, wrist=wpositive, fatherId=fReference[0]}
  [339] = {x=208.852, y=-30.028, z=44, rx=180, rz=-83.182, shoulder=lefty, elbow=epositive, wrist=wpositive, fatherId=fReference[0]}
  [340] = {x=210.045, y=-20.057, z=44, rx=180, rz=-85.909, shoulder=lefty, elbow=epositive, wrist=wpositive, fatherId=fReference[0]}
  [341] = {x=210.761, y=-10.04, z=44, rx=180, rz=-88.636, shoulder=lefty, elbow=epositive, wrist=wpositive, fatherId=fReference[0]}
  [342] = {x=211, z=44, rx=-180, rz=-91.364, shoulder=lefty, elbow=epositive, wrist=wpositive, fatherId=fReference[0]}
  [343] = {x=210.761, y=10.04, z=44, rx=-180, rz=-94.091, shoulder=lefty, elbow=epositive, wrist=wpositive, fatherId=fReference[0]}
  [344] = {x=210.045, y=20.057, z=44, rx=-180, rz=-96.818, shoulder=lefty, elbow=epositive, wrist=wpositive, fatherId=fReference[0]}
  [345] = {x=208.852, y=30.028, z=44, rx=-180, rz=-99.545, shoulder=lefty, elbow=epositive, wrist=wpositive, fatherId=fReference[0]}
  [346] = {x=207.187, y=39.932, z=44, rx=-180, rz=-102.273, shoulder=lefty, elbow=epositive, wrist=wpositive, fatherId=fReference[0]}
  [347] = {x=205.052, y=49.745, z=44, rx=-180, rz=-105, shoulder=lefty, elbow=epositive, wrist=wpositive, fatherId=fReference[0]}
  [348] = {x=202.453, y=59.446, z=44, rx=-180, rz=-107.727, shoulder=lefty, elbow=epositive, wrist=wpositive, fatherId=fReference[0]}
  [349] = {x=199.395, y=69.011, z=44, rx=-180, rz=-110.455, shoulder=lefty, elbow=epositive, wrist=wpositive, fatherId=fReference[0]}
  [350] = {x=195.886, y=78.421, z=44, rx=-180, rz=-113.182, shoulder=lefty, elbow=epositive, wrist=wpositive, fatherId=fReference[0]}
  [351] = {x=191.932, y=87.653, z=44, rx=-180, rz=-115.909, shoulder=lefty, elbow=epositive, wrist=wpositive, fatherId=fReference[0]}
  [352] = {x=187.544, y=96.686, z=44, rx=-180, rz=-118.636, shoulder=lefty, elbow=epositive, wrist=wpositive, fatherId=fReference[0]}
  [353] = {x=182.731, y=105.5, z=44, rx=-180, rz=-121.364, shoulder=lefty, elbow=epositive, wrist=wpositive, fatherId=fReference[0]}
  [354] = {x=177.505, y=114.075, z=44, rx=-180, rz=-124.091, shoulder=lefty, elbow=epositive, wrist=wpositive, fatherId=fReference[0]}
  [355] = {x=171.876, y=122.392, z=44, rx=-180, rz=-126.818, shoulder=lefty, elbow=epositive, wrist=wpositive, fatherId=fReference[0]}
  [356] = {x=165.857, y=130.432, z=44, rx=-180, rz=-129.545, shoulder=lefty, elbow=epositive, wrist=wpositive, fatherId=fReference[0]}
  [357] = {x=159.463, y=138.176, z=44, rx=-180, rz=-132.273, shoulder=lefty, elbow=epositive, wrist=wpositive, fatherId=fReference[0]}
  [358] = {x=152.708, y=145.607, z=44, rx=-180, rz=-135, shoulder=lefty, elbow=epositive, wrist=wpositive, fatherId=fReference[0]}
  [359] = {x=145.607, y=152.708, z=44, rx=-180, rz=-137.727, shoulder=lefty, elbow=epositive, wrist=wpositive, fatherId=fReference[0]}
  [360] = {x=138.176, y=159.463, z=44, rx=180, rz=-140.455, shoulder=lefty, elbow=epositive, wrist=wpositive, fatherId=fReference[0]}
  [361] = {x=130.432, y=165.857, z=44, rx=-180, rz=-143.182, shoulder=lefty, elbow=epositive, wrist=wpositive, fatherId=fReference[0]}
  [362] = {x=122.392, y=171.876, z=44, rx=-180, rz=-145.909, shoulder=lefty, elbow=epositive, wrist=wpositive, fatherId=fReference[0]}
  [363] = {x=114.075, y=177.505, z=44, rx=-180, rz=-148.636, shoulder=lefty, elbow=epositive, wrist=wpositive, fatherId=fReference[0]}
  [364] = {x=105.5, y=182.731, z=44, rx=-180, rz=-151.364, shoulder=lefty, elbow=epositive, wrist=wpositive, fatherId=fReference[0]}
  [365] = {x=96.686, y=187.544, z=44, rx=180, rz=-154.091, shoulder=lefty, elbow=epositive, wrist=wpositive, fatherId=fReference[0]}
  [366] = {x=87.653, y=191.932, z=44, rx=-180, rz=-156.818, shoulder=lefty, elbow=epositive, wrist=wpositive, fatherId=fReference[0]}
  [367] = {x=78.421, y=195.886, z=44, rx=180, rz=-159.545, shoulder=lefty, elbow=epositive, wrist=wpositive, fatherId=fReference[0]}
  [368] = {x=69.011, y=199.395, z=44, rx=-180, rz=-162.273, shoulder=lefty, elbow=epositive, wrist=wpositive, fatherId=fReference[0]}
  [369] = {x=59.446, y=202.453, z=44, rx=-180, rz=-165, shoulder=lefty, elbow=epositive, wrist=wpositive, fatherId=fReference[0]}
  [370] = {x=49.745, y=205.052, z=44, rx=180, rz=-167.727, shoulder=lefty, elbow=epositive, wrist=wpositive, fatherId=fReference[0]}
  [371] = {x=39.932, y=207.187, z=44, rx=180, rz=-170.455, shoulder=lefty, elbow=epositive, wrist=wpositive, fatherId=fReference[0]}
  [372] = {x=30.028, y=208.852, z=44, rx=-180, rz=-173.182, shoulder=lefty, elbow=epositive, wrist=wpositive, fatherId=fReference[0]}
  [373] = {x=20.057, y=210.045, z=44, rx=180, rz=-175.909, shoulder=lefty, elbow=epositive, wrist=wpositive, fatherId=fReference[0]}
  [374] = {x=10.04, y=210.761, z=44, rx=180, rz=-178.636, shoulder=lefty, elbow=epositive, wrist=wpositive, fatherId=fReference[0]}
  [375] = {y=211, z=44, rx=-180, rz=178.636, shoulder=lefty, elbow=epositive, wrist=wpositive, fatherId=fReference[0]}
  [376] = {x=-10.04, y=210.761, z=44, rx=-180, rz=175.909, shoulder=lefty, elbow=epositive, wrist=wpositive, fatherId=fReference[0]}
  [377] = {x=-20.057, y=210.045, z=44, rx=-180, rz=173.182, shoulder=lefty, elbow=epositive, wrist=wpositive, fatherId=fReference[0]}
  [378] = {x=-30.028, y=208.852, z=44, rx=180, rz=170.455, shoulder=lefty, elbow=epositive, wrist=wpositive, fatherId=fReference[0]}
  [379] = {x=-39.932, y=207.187, z=44, rx=180, rz=167.727, shoulder=lefty, elbow=epositive, wrist=wpositive, fatherId=fReference[0]}
  [380] = {x=-49.745, y=205.052, z=44, rx=180, rz=165, shoulder=lefty, elbow=epositive, wrist=wpositive, fatherId=fReference[0]}
  [381] = {x=-59.446, y=202.453, z=44, rx=-180, rz=162.273, shoulder=lefty, elbow=epositive, wrist=wpositive, fatherId=fReference[0]}
  [382] = {x=-69.011, y=199.395, z=44, rx=180, rz=159.545, shoulder=lefty, elbow=epositive, wrist=wpositive, fatherId=fReference[0]}
  [383] = {x=-78.421, y=195.886, z=44, rx=180, rz=156.818, shoulder=lefty, elbow=epositive, wrist=wpositive, fatherId=fReference[0]}
  [384] = {x=-87.653, y=191.932, z=44, rx=180, rz=154.091, shoulder=lefty, elbow=epositive, wrist=wpositive, fatherId=fReference[0]}
  [385] = {x=-96.686, y=187.544, z=44, rx=180, rz=151.364, shoulder=lefty, elbow=epositive, wrist=wpositive, fatherId=fReference[0]}
  [386] = {x=-105.5, y=182.731, z=44, rx=180, rz=148.636, shoulder=lefty, elbow=epositive, wrist=wpositive, fatherId=fReference[0]}
  [387] = {x=-114.075, y=177.505, z=44, rx=180, rz=145.909, shoulder=lefty, elbow=epositive, wrist=wpositive, fatherId=fReference[0]}
  [388] = {x=-122.392, y=171.876, z=44, rx=180, rz=143.182, shoulder=lefty, elbow=epositive, wrist=wpositive, fatherId=fReference[0]}
  [389] = {x=-130.432, y=165.857, z=44, rx=180, rz=140.455, shoulder=lefty, elbow=epositive, wrist=wpositive, fatherId=fReference[0]}
  [390] = {x=-138.176, y=159.463, z=44, rx=-180, rz=137.727, shoulder=lefty, elbow=epositive, wrist=wpositive, fatherId=fReference[0]}
  [391] = {x=-145.607, y=152.708, z=44, rx=-180, rz=135, shoulder=lefty, elbow=epositive, wrist=wpositive, fatherId=fReference[0]}
  [392] = {x=-152.708, y=145.607, z=44, rx=180, rz=132.273, shoulder=lefty, elbow=epositive, wrist=wpositive, fatherId=fReference[0]}
  [393] = {x=-159.463, y=138.176, z=44, rx=180, rz=129.545, shoulder=lefty, elbow=epositive, wrist=wpositive, fatherId=fReference[0]}
  [394] = {x=-165.857, y=130.432, z=44, rx=180, rz=126.818, shoulder=lefty, elbow=epositive, wrist=wpositive, fatherId=fReference[0]}
  [395] = {x=-171.876, y=122.392, z=44, rx=180, rz=124.091, shoulder=lefty, elbow=epositive, wrist=wpositive, fatherId=fReference[0]}
  [396] = {x=-177.505, y=114.075, z=44, rx=-180, rz=121.364, shoulder=lefty, elbow=epositive, wrist=wpositive, fatherId=fReference[0]}
  [397] = {x=-182.731, y=105.5, z=44, rx=180, rz=118.636, shoulder=lefty, elbow=epositive, wrist=wpositive, fatherId=fReference[0]}
  [398] = {x=-187.544, y=96.686, z=44, rx=180, rz=115.909, shoulder=lefty, elbow=epositive, wrist=wpositive, fatherId=fReference[0]}
  [399] = {x=-191.932, y=87.653, z=44, rx=180, rz=113.182, shoulder=lefty, elbow=epositive, wrist=wpositive, fatherId=fReference[0]}
  [400] = {x=-195.886, y=78.421, z=44, rx=180, rz=110.455, shoulder=lefty, elbow=epositive, wrist=wpositive, fatherId=fReference[0]}
  [401] = {x=-199.395, y=69.011, z=44, rx=180, rz=107.727, shoulder=lefty, elbow=epositive, wrist=wpositive, fatherId=fReference[0]}
  [402] = {x=-202.453, y=59.446, z=44, rx=180, rz=105, shoulder=lefty, elbow=epositive, wrist=wpositive, fatherId=fReference[0]}
  [403] = {x=-205.052, y=49.745, z=44, rx=180, rz=102.273, shoulder=lefty, elbow=epositive, wrist=wpositive, fatherId=fReference[0]}
  [404] = {x=-207.187, y=39.932, z=44, rx=180, rz=99.545, shoulder=lefty, elbow=epositive, wrist=wpositive, fatherId=fReference[0]}
  [405] = {x=-208.852, y=30.028, z=44, rx=180, rz=96.818, shoulder=lefty, elbow=epositive, wrist=wpositive, fatherId=fReference[0]}
  [406] = {x=-210.045, y=20.057, z=44, rx=180, rz=94.091, shoulder=lefty, elbow=epositive, wrist=wpositive, fatherId=fReference[0]}
  [407] = {x=-210.761, y=10.04, z=44, rx=180, rz=91.364, shoulder=lefty, elbow=epositive, wrist=wpositive, fatherId=fReference[0]}
  [408] = {x=-211, z=44, rx=180, rz=91.364, shoulder=lefty, elbow=epositive, wrist=wpositive, fatherId=fReference[0]}
  [409] = {x=-211, z=44, rx=180, rz=91.364, shoulder=lefty, elbow=epositive, wrist=wpositive, fatherId=fReference[0]}
  [410] = {x=-211, z=144, rx=180, rz=91.364, shoulder=lefty, elbow=epositive, wrist=wpositive, fatherId=fReference[0]}
  [411] = {x=-211, z=166, rx=180, rz=91.364, shoulder=lefty, elbow=epositive, wrist=wpositive, fatherId=fReference[0]}
  [412] = {x=-211, z=66, rx=180, rz=91.364, shoulder=lefty, elbow=epositive, wrist=wpositive, fatherId=fReference[0]}
  [413] = {x=-211, z=66, rx=180, rz=91.364, shoulder=lefty, elbow=epositive, wrist=wpositive, fatherId=fReference[0]}
  [414] = {x=-210.761, y=10.04, z=66, rx=180, rz=94.091, shoulder=lefty, elbow=epositive, wrist=wpositive, fatherId=fReference[0]}
  [415] = {x=-210.045, y=20.057, z=66, rx=180, rz=96.818, shoulder=lefty, elbow=epositive, wrist=wpositive, fatherId=fReference[0]}
  [416] = {x=-208.852, y=30.028, z=66, rx=180, rz=99.545, shoulder=lefty, elbow=epositive, wrist=wpositive, fatherId=fReference[0]}
  [417] = {x=-207.187, y=39.932, z=66, rx=180, rz=102.273, shoulder=lefty, elbow=epositive, wrist=wpositive, fatherId=fReference[0]}
  [418] = {x=-205.052, y=49.745, z=66, rx=180, rz=105, shoulder=lefty, elbow=epositive, wrist=wpositive, fatherId=fReference[0]}
  [419] = {x=-202.453, y=59.446, z=66, rx=180, rz=107.727, shoulder=lefty, elbow=epositive, wrist=wpositive, fatherId=fReference[0]}
  [420] = {x=-199.395, y=69.011, z=66, rx=180, rz=110.455, shoulder=lefty, elbow=epositive, wrist=wpositive, fatherId=fReference[0]}
  [421] = {x=-195.886, y=78.421, z=66, rx=180, rz=113.182, shoulder=lefty, elbow=epositive, wrist=wpositive, fatherId=fReference[0]}
  [422] = {x=-191.932, y=87.653, z=66, rx=180, rz=115.909, shoulder=lefty, elbow=epositive, wrist=wpositive, fatherId=fReference[0]}
  [423] = {x=-187.544, y=96.686, z=66, rx=-180, rz=118.636, shoulder=lefty, elbow=epositive, wrist=wpositive, fatherId=fReference[0]}
  [424] = {x=-182.731, y=105.5, z=66, rx=180, rz=121.364, shoulder=lefty, elbow=epositive, wrist=wpositive, fatherId=fReference[0]}
  [425] = {x=-177.505, y=114.075, z=66, rx=180, rz=124.091, shoulder=lefty, elbow=epositive, wrist=wpositive, fatherId=fReference[0]}
  [426] = {x=-171.876, y=122.392, z=66, rx=-180, rz=126.818, shoulder=lefty, elbow=epositive, wrist=wpositive, fatherId=fReference[0]}
  [427] = {x=-165.857, y=130.432, z=66, rx=180, rz=129.545, shoulder=lefty, elbow=epositive, wrist=wpositive, fatherId=fReference[0]}
  [428] = {x=-159.463, y=138.176, z=66, rx=180, rz=132.273, shoulder=lefty, elbow=epositive, wrist=wpositive, fatherId=fReference[0]}
  [429] = {x=-152.708, y=145.607, z=66, rx=180, rz=135, shoulder=lefty, elbow=epositive, wrist=wpositive, fatherId=fReference[0]}
  [430] = {x=-145.607, y=152.708, z=66, rx=180, rz=137.727, shoulder=lefty, elbow=epositive, wrist=wpositive, fatherId=fReference[0]}
  [431] = {x=-138.176, y=159.463, z=66, rx=-180, rz=140.455, shoulder=lefty, elbow=epositive, wrist=wpositive, fatherId=fReference[0]}
  [432] = {x=-130.432, y=165.857, z=66, rx=180, rz=143.182, shoulder=lefty, elbow=epositive, wrist=wpositive, fatherId=fReference[0]}
  [433] = {x=-122.392, y=171.876, z=66, rx=-180, rz=145.909, shoulder=lefty, elbow=epositive, wrist=wpositive, fatherId=fReference[0]}
  [434] = {x=-114.075, y=177.505, z=66, rx=180, rz=148.636, shoulder=lefty, elbow=epositive, wrist=wpositive, fatherId=fReference[0]}
  [435] = {x=-105.5, y=182.731, z=66, rx=-180, rz=151.364, shoulder=lefty, elbow=epositive, wrist=wpositive, fatherId=fReference[0]}
  [436] = {x=-96.686, y=187.544, z=66, rx=-180, rz=154.091, shoulder=lefty, elbow=epositive, wrist=wpositive, fatherId=fReference[0]}
  [437] = {x=-87.653, y=191.932, z=66, rx=180, rz=156.818, shoulder=lefty, elbow=epositive, wrist=wpositive, fatherId=fReference[0]}
  [438] = {x=-78.421, y=195.886, z=66, rx=180, rz=159.545, shoulder=lefty, elbow=epositive, wrist=wpositive, fatherId=fReference[0]}
  [439] = {x=-69.011, y=199.395, z=66, rx=180, rz=162.273, shoulder=lefty, elbow=epositive, wrist=wpositive, fatherId=fReference[0]}
  [440] = {x=-59.446, y=202.453, z=66, rx=180, rz=165, shoulder=lefty, elbow=epositive, wrist=wpositive, fatherId=fReference[0]}
  [441] = {x=-49.745, y=205.052, z=66, rx=180, rz=167.727, shoulder=lefty, elbow=epositive, wrist=wpositive, fatherId=fReference[0]}
  [442] = {x=-39.932, y=207.187, z=66, rx=-180, rz=170.455, shoulder=lefty, elbow=epositive, wrist=wpositive, fatherId=fReference[0]}
  [443] = {x=-30.028, y=208.852, z=66, rx=-180, rz=173.182, shoulder=lefty, elbow=epositive, wrist=wpositive, fatherId=fReference[0]}
  [444] = {x=-20.057, y=210.045, z=66, rx=-180, rz=175.909, shoulder=lefty, elbow=epositive, wrist=wpositive, fatherId=fReference[0]}
  [445] = {x=-10.04, y=210.761, z=66, rx=180, rz=178.636, shoulder=lefty, elbow=epositive, wrist=wpositive, fatherId=fReference[0]}
  [446] = {y=211, z=66, rx=180, rz=-178.636, shoulder=lefty, elbow=epositive, wrist=wpositive, fatherId=fReference[0]}
  [447] = {x=10.04, y=210.761, z=66, rx=-180, rz=-175.909, shoulder=lefty, elbow=epositive, wrist=wpositive, fatherId=fReference[0]}
  [448] = {x=20.057, y=210.045, z=66, rx=-180, rz=-173.182, shoulder=lefty, elbow=epositive, wrist=wpositive, fatherId=fReference[0]}
  [449] = {x=30.028, y=208.852, z=66, rx=-180, rz=-170.455, shoulder=lefty, elbow=epositive, wrist=wpositive, fatherId=fReference[0]}
  [450] = {x=39.932, y=207.187, z=66, rx=-180, rz=-167.727, shoulder=lefty, elbow=epositive, wrist=wpositive, fatherId=fReference[0]}
  [451] = {x=49.745, y=205.052, z=66, rx=-180, rz=-165, shoulder=lefty, elbow=epositive, wrist=wpositive, fatherId=fReference[0]}
  [452] = {x=59.446, y=202.453, z=66, rx=180, rz=-162.273, shoulder=lefty, elbow=epositive, wrist=wpositive, fatherId=fReference[0]}
  [453] = {x=69.011, y=199.395, z=66, rx=-180, rz=-159.545, shoulder=lefty, elbow=epositive, wrist=wpositive, fatherId=fReference[0]}
  [454] = {x=78.421, y=195.886, z=66, rx=-180, rz=-156.818, shoulder=lefty, elbow=epositive, wrist=wpositive, fatherId=fReference[0]}
  [455] = {x=87.653, y=191.932, z=66, rx=-180, rz=-154.091, shoulder=lefty, elbow=epositive, wrist=wpositive, fatherId=fReference[0]}
  [456] = {x=96.686, y=187.544, z=66, rx=-180, rz=-151.364, shoulder=lefty, elbow=epositive, wrist=wpositive, fatherId=fReference[0]}
  [457] = {x=105.5, y=182.731, z=66, rx=-180, rz=-148.636, shoulder=lefty, elbow=epositive, wrist=wpositive, fatherId=fReference[0]}
  [458] = {x=114.075, y=177.505, z=66, rx=180, rz=-145.909, shoulder=lefty, elbow=epositive, wrist=wpositive, fatherId=fReference[0]}
  [459] = {x=122.392, y=171.876, z=66, rx=-180, rz=-143.182, shoulder=lefty, elbow=epositive, wrist=wpositive, fatherId=fReference[0]}
  [460] = {x=130.432, y=165.857, z=66, rx=-180, rz=-140.455, shoulder=lefty, elbow=epositive, wrist=wpositive, fatherId=fReference[0]}
  [461] = {x=138.176, y=159.463, z=66, rx=-180, rz=-137.727, shoulder=lefty, elbow=epositive, wrist=wpositive, fatherId=fReference[0]}
  [462] = {x=145.607, y=152.708, z=66, rx=-180, rz=-135, shoulder=lefty, elbow=epositive, wrist=wpositive, fatherId=fReference[0]}
  [463] = {x=152.708, y=145.607, z=66, rx=-180, rz=-132.273, shoulder=lefty, elbow=epositive, wrist=wpositive, fatherId=fReference[0]}
  [464] = {x=159.463, y=138.176, z=66, rx=-180, rz=-129.545, shoulder=lefty, elbow=epositive, wrist=wpositive, fatherId=fReference[0]}
  [465] = {x=165.857, y=130.432, z=66, rx=-180, rz=-126.818, shoulder=lefty, elbow=epositive, wrist=wpositive, fatherId=fReference[0]}
  [466] = {x=171.876, y=122.392, z=66, rx=-180, rz=-124.091, shoulder=lefty, elbow=epositive, wrist=wpositive, fatherId=fReference[0]}
  [467] = {x=177.505, y=114.075, z=66, rx=-180, rz=-121.364, shoulder=lefty, elbow=epositive, wrist=wpositive, fatherId=fReference[0]}
  [468] = {x=182.731, y=105.5, z=66, rx=-180, rz=-118.636, shoulder=lefty, elbow=epositive, wrist=wpositive, fatherId=fReference[0]}
  [469] = {x=187.544, y=96.686, z=66, rx=-180, rz=-115.909, shoulder=lefty, elbow=epositive, wrist=wpositive, fatherId=fReference[0]}
  [470] = {x=191.932, y=87.653, z=66, rx=-180, rz=-113.182, shoulder=lefty, elbow=epositive, wrist=wpositive, fatherId=fReference[0]}
  [471] = {x=195.886, y=78.421, z=66, rx=-180, rz=-110.455, shoulder=lefty, elbow=epositive, wrist=wpositive, fatherId=fReference[0]}
  [472] = {x=199.395, y=69.011, z=66, rx=-180, rz=-107.727, shoulder=lefty, elbow=epositive, wrist=wpositive, fatherId=fReference[0]}
  [473] = {x=202.453, y=59.446, z=66, rx=-180, rz=-105, shoulder=lefty, elbow=epositive, wrist=wpositive, fatherId=fReference[0]}
  [474] = {x=205.052, y=49.745, z=66, rx=-180, rz=-102.273, shoulder=lefty, elbow=epositive, wrist=wpositive, fatherId=fReference[0]}
  [475] = {x=207.187, y=39.932, z=66, rx=-180, rz=-99.545, shoulder=lefty, elbow=epositive, wrist=wpositive, fatherId=fReference[0]}
  [476] = {x=208.852, y=30.028, z=66, rx=-180, rz=-96.818, shoulder=lefty, elbow=epositive, wrist=wpositive, fatherId=fReference[0]}
  [477] = {x=210.045, y=20.057, z=66, rx=-180, rz=-94.091, shoulder=lefty, elbow=epositive, wrist=wpositive, fatherId=fReference[0]}
  [478] = {x=210.761, y=10.04, z=66, rx=-180, rz=-91.364, shoulder=lefty, elbow=epositive, wrist=wpositive, fatherId=fReference[0]}
  [479] = {x=211, z=66, rx=180, rz=-88.636, shoulder=lefty, elbow=epositive, wrist=wpositive, fatherId=fReference[0]}
  [480] = {x=210.761, y=-10.04, z=66, rx=180, rz=-85.909, shoulder=lefty, elbow=epositive, wrist=wpositive, fatherId=fReference[0]}
  [481] = {x=210.045, y=-20.057, z=66, rx=180, rz=-83.182, shoulder=lefty, elbow=epositive, wrist=wpositive, fatherId=fReference[0]}
  [482] = {x=208.852, y=-30.028, z=66, rx=180, rz=-80.455, shoulder=lefty, elbow=epositive, wrist=wpositive, fatherId=fReference[0]}
  [483] = {x=207.187, y=-39.932, z=66, rx=180, rz=-77.727, shoulder=lefty, elbow=epositive, wrist=wpositive, fatherId=fReference[0]}
  [484] = {x=205.052, y=-49.745, z=66, rx=180, rz=-75, shoulder=lefty, elbow=epositive, wrist=wpositive, fatherId=fReference[0]}
  [485] = {x=202.453, y=-59.446, z=66, rx=180, rz=-72.273, shoulder=lefty, elbow=epositive, wrist=wpositive, fatherId=fReference[0]}
  [486] = {x=199.395, y=-69.011, z=66, rx=180, rz=-69.545, shoulder=lefty, elbow=epositive, wrist=wpositive, fatherId=fReference[0]}
  [487] = {x=195.886, y=-78.421, z=66, rx=180, rz=-66.818, shoulder=lefty, elbow=epositive, wrist=wpositive, fatherId=fReference[0]}
  [488] = {x=191.932, y=-87.653, z=66, rx=-180, rz=-64.091, shoulder=lefty, elbow=epositive, wrist=wpositive, fatherId=fReference[0]}
  [489] = {x=187.544, y=-96.686, z=66, rx=180, rz=-61.364, shoulder=lefty, elbow=epositive, wrist=wpositive, fatherId=fReference[0]}
  [490] = {x=182.731, y=-105.5, z=66, rx=180, rz=-58.636, shoulder=lefty, elbow=epositive, wrist=wpositive, fatherId=fReference[0]}
  [491] = {x=177.505, y=-114.075, z=66, rx=180, rz=-55.909, shoulder=lefty, elbow=epositive, wrist=wpositive, fatherId=fReference[0]}
  [492] = {x=171.876, y=-122.392, z=66, rx=180, rz=-53.182, shoulder=lefty, elbow=epositive, wrist=wpositive, fatherId=fReference[0]}
  [493] = {x=165.857, y=-130.432, z=66, rx=-180, rz=-50.455, shoulder=lefty, elbow=epositive, wrist=wpositive, fatherId=fReference[0]}
  [494] = {x=159.463, y=-138.176, z=66, rx=-180, rz=-47.727, shoulder=lefty, elbow=epositive, wrist=wpositive, fatherId=fReference[0]}
  [495] = {x=152.708, y=-145.607, z=66, rx=-180, rz=-45, shoulder=lefty, elbow=epositive, wrist=wpositive, fatherId=fReference[0]}
  [496] = {x=145.607, y=-152.708, z=66, rx=180, rz=-42.273, shoulder=lefty, elbow=epositive, wrist=wpositive, fatherId=fReference[0]}
  [497] = {x=138.176, y=-159.463, z=66, rx=180, rz=-39.545, shoulder=lefty, elbow=epositive, wrist=wpositive, fatherId=fReference[0]}
  [498] = {x=130.432, y=-165.857, z=66, rx=180, rz=-36.818, shoulder=lefty, elbow=epositive, wrist=wpositive, fatherId=fReference[0]}
  [499] = {x=122.392, y=-171.876, z=66, rx=180, rz=-34.091, shoulder=lefty, elbow=epositive, wrist=wpositive, fatherId=fReference[0]}
  [500] = {x=114.075, y=-177.505, z=66, rx=180, rz=-31.364, shoulder=lefty, elbow=epositive, wrist=wpositive, fatherId=fReference[0]}
  [501] = {x=105.5, y=-182.731, z=66, rx=-180, rz=-28.636, shoulder=lefty, elbow=epositive, wrist=wpositive, fatherId=fReference[0]}
  [502] = {x=96.686, y=-187.544, z=66, rx=180, rz=-25.909, shoulder=lefty, elbow=epositive, wrist=wpositive, fatherId=fReference[0]}
  [503] = {x=87.653, y=-191.932, z=66, rx=-180, rz=-23.182, shoulder=lefty, elbow=epositive, wrist=wpositive, fatherId=fReference[0]}
  [504] = {x=78.421, y=-195.886, z=66, rx=180, rz=-20.455, shoulder=lefty, elbow=epositive, wrist=wpositive, fatherId=fReference[0]}
  [505] = {x=69.011, y=-199.395, z=66, rx=180, rz=-17.727, shoulder=lefty, elbow=epositive, wrist=wpositive, fatherId=fReference[0]}
  [506] = {x=59.446, y=-202.453, z=66, rx=-180, rz=-15, shoulder=lefty, elbow=epositive, wrist=wpositive, fatherId=fReference[0]}
  [507] = {x=49.745, y=-205.052, z=66, rx=-180, rz=-12.273, shoulder=lefty, elbow=epositive, wrist=wpositive, fatherId=fReference[0]}
  [508] = {x=39.932, y=-207.187, z=66, rx=-180, rz=-9.545, shoulder=lefty, elbow=epositive, wrist=wpositive, fatherId=fReference[0]}
  [509] = {x=30.028, y=-208.852, z=66, rx=-180, rz=-6.818, shoulder=lefty, elbow=epositive, wrist=wpositive, fatherId=fReference[0]}
  [510] = {x=20.057, y=-210.045, z=66, rx=180, rz=-4.091, shoulder=lefty, elbow=epositive, wrist=wpositive, fatherId=fReference[0]}
  [511] = {x=10.04, y=-210.761, z=66, rx=-180, rz=-1.364, shoulder=lefty, elbow=epositive, wrist=wpositive, fatherId=fReference[0]}
  [512] = {y=-211, z=66, rx=180, rz=1.364, shoulder=lefty, elbow=epositive, wrist=wpositive, fatherId=fReference[0]}
  [513] = {x=-10.04, y=-210.761, z=66, rx=180, rz=4.091, shoulder=lefty, elbow=epositive, wrist=wpositive, fatherId=fReference[0]}
  [514] = {x=-20.057, y=-210.045, z=66, rx=-180, rz=6.818, shoulder=lefty, elbow=epositive, wrist=wpositive, fatherId=fReference[0]}
  [515] = {x=-30.028, y=-208.852, z=66, rx=-180, rz=9.545, shoulder=lefty, elbow=epositive, wrist=wpositive, fatherId=fReference[0]}
  [516] = {x=-39.932, y=-207.187, z=66, rx=-180, rz=12.273, shoulder=lefty, elbow=epositive, wrist=wpositive, fatherId=fReference[0]}
  [517] = {x=-49.745, y=-205.052, z=66, rx=180, rz=15, shoulder=lefty, elbow=epositive, wrist=wpositive, fatherId=fReference[0]}
  [518] = {x=-59.446, y=-202.453, z=66, rx=180, rz=17.727, shoulder=lefty, elbow=epositive, wrist=wpositive, fatherId=fReference[0]}
  [519] = {x=-69.011, y=-199.395, z=66, rx=-180, rz=20.455, shoulder=lefty, elbow=epositive, wrist=wpositive, fatherId=fReference[0]}
  [520] = {x=-78.421, y=-195.886, z=66, rx=-180, rz=23.182, shoulder=lefty, elbow=epositive, wrist=wpositive, fatherId=fReference[0]}
  [521] = {x=-87.653, y=-191.932, z=66, rx=180, rz=25.909, shoulder=lefty, elbow=epositive, wrist=wpositive, fatherId=fReference[0]}
  [522] = {x=-96.686, y=-187.544, z=66, rx=-180, rz=28.636, shoulder=lefty, elbow=epositive, wrist=wpositive, fatherId=fReference[0]}
  [523] = {x=-105.5, y=-182.731, z=66, rx=-180, rz=31.364, shoulder=lefty, elbow=epositive, wrist=wpositive, fatherId=fReference[0]}
  [524] = {x=-114.075, y=-177.505, z=66, rx=-180, rz=34.091, shoulder=lefty, elbow=epositive, wrist=wpositive, fatherId=fReference[0]}
  [525] = {x=-122.392, y=-171.876, z=66, rx=180, rz=36.818, shoulder=lefty, elbow=epositive, wrist=wpositive, fatherId=fReference[0]}
  [526] = {x=-130.432, y=-165.857, z=66, rx=180, rz=39.545, shoulder=lefty, elbow=epositive, wrist=wpositive, fatherId=fReference[0]}
  [527] = {x=-138.176, y=-159.463, z=66, rx=-180, rz=42.273, shoulder=lefty, elbow=epositive, wrist=wpositive, fatherId=fReference[0]}
  [528] = {x=-145.607, y=-152.708, z=66, rx=-180, rz=45, shoulder=lefty, elbow=epositive, wrist=wpositive, fatherId=fReference[0]}
  [529] = {x=-152.708, y=-145.607, z=66, rx=-180, rz=47.727, shoulder=lefty, elbow=epositive, wrist=wpositive, fatherId=fReference[0]}
  [530] = {x=-159.463, y=-138.176, z=66, rx=-180, rz=50.455, shoulder=lefty, elbow=epositive, wrist=wpositive, fatherId=fReference[0]}
  [531] = {x=-165.857, y=-130.432, z=66, rx=-180, rz=53.182, shoulder=lefty, elbow=epositive, wrist=wpositive, fatherId=fReference[0]}
  [532] = {x=-171.876, y=-122.392, z=66, rx=-180, rz=55.909, shoulder=lefty, elbow=epositive, wrist=wpositive, fatherId=fReference[0]}
  [533] = {x=-177.505, y=-114.075, z=66, rx=-180, rz=58.636, shoulder=lefty, elbow=epositive, wrist=wpositive, fatherId=fReference[0]}
  [534] = {x=-182.731, y=-105.5, z=66, rx=-180, rz=61.364, shoulder=lefty, elbow=epositive, wrist=wpositive, fatherId=fReference[0]}
  [535] = {x=-187.544, y=-96.686, z=66, rx=-180, rz=64.091, shoulder=lefty, elbow=epositive, wrist=wpositive, fatherId=fReference[0]}
  [536] = {x=-191.932, y=-87.653, z=66, rx=-180, rz=66.818, shoulder=lefty, elbow=epositive, wrist=wpositive, fatherId=fReference[0]}
  [537] = {x=-195.886, y=-78.421, z=66, rx=-180, rz=69.545, shoulder=lefty, elbow=epositive, wrist=wpositive, fatherId=fReference[0]}
  [538] = {x=-199.395, y=-69.011, z=66, rx=-180, rz=72.273, shoulder=lefty, elbow=epositive, wrist=wpositive, fatherId=fReference[0]}
  [539] = {x=-202.453, y=-59.446, z=66, rx=-180, rz=75, shoulder=lefty, elbow=epositive, wrist=wpositive, fatherId=fReference[0]}
  [540] = {x=-205.052, y=-49.745, z=66, rx=-180, rz=77.727, shoulder=lefty, elbow=epositive, wrist=wpositive, fatherId=fReference[0]}
  [541] = {x=-207.187, y=-39.932, z=66, rx=-180, rz=80.455, shoulder=lefty, elbow=epositive, wrist=wpositive, fatherId=fReference[0]}
  [542] = {x=-208.852, y=-30.028, z=66, rx=-180, rz=83.182, shoulder=lefty, elbow=epositive, wrist=wpositive, fatherId=fReference[0]}
  [543] = {x=-210.045, y=-20.057, z=66, rx=-180, rz=85.909, shoulder=lefty, elbow=epositive, wrist=wpositive, fatherId=fReference[0]}
  [544] = {x=-210.761, y=-10.04, z=66, rx=-180, rz=88.636, shoulder=lefty, elbow=epositive, wrist=wpositive, fatherId=fReference[0]}
  [545] = {x=-211, z=66, rx=-180, rz=88.636, shoulder=lefty, elbow=epositive, wrist=wpositive, fatherId=fReference[0]}
  [546] = {x=-211, z=66, rx=-180, rz=88.636, shoulder=lefty, elbow=epositive, wrist=wpositive, fatherId=fReference[0]}
  [547] = {x=-211, z=166, rx=-180, rz=88.636, shoulder=lefty, elbow=epositive, wrist=wpositive, fatherId=fReference[0]}
  [548] = {x=-211, z=188, rx=-180, rz=88.636, shoulder=lefty, elbow=epositive, wrist=wpositive, fatherId=fReference[0]}
  [549] = {x=-211, z=88, rx=-180, rz=88.636, shoulder=lefty, elbow=epositive, wrist=wpositive, fatherId=fReference[0]}
  [550] = {x=-211, z=88, rx=-180, rz=88.636, shoulder=lefty, elbow=epositive, wrist=wpositive, fatherId=fReference[0]}
  [551] = {x=-210.761, y=-10.04, z=88, rx=-180, rz=85.909, shoulder=lefty, elbow=epositive, wrist=wpositive, fatherId=fReference[0]}
  [552] = {x=-210.045, y=-20.057, z=88, rx=-180, rz=83.182, shoulder=lefty, elbow=epositive, wrist=wpositive, fatherId=fReference[0]}
  [553] = {x=-208.852, y=-30.028, z=88, rx=-180, rz=80.455, shoulder=lefty, elbow=epositive, wrist=wpositive, fatherId=fReference[0]}
  [554] = {x=-207.187, y=-39.932, z=88, rx=-180, rz=77.727, shoulder=lefty, elbow=epositive, wrist=wpositive, fatherId=fReference[0]}
  [555] = {x=-205.052, y=-49.745, z=88, rx=-180, rz=75, shoulder=lefty, elbow=epositive, wrist=wpositive, fatherId=fReference[0]}
  [556] = {x=-202.453, y=-59.446, z=88, rx=-180, rz=72.273, shoulder=lefty, elbow=epositive, wrist=wpositive, fatherId=fReference[0]}
  [557] = {x=-199.395, y=-69.011, z=88, rx=-180, rz=69.545, shoulder=lefty, elbow=epositive, wrist=wpositive, fatherId=fReference[0]}
  [558] = {x=-195.886, y=-78.421, z=88, rx=-180, rz=66.818, shoulder=lefty, elbow=epositive, wrist=wpositive, fatherId=fReference[0]}
  [559] = {x=-191.932, y=-87.653, z=88, rx=-180, rz=64.091, shoulder=lefty, elbow=epositive, wrist=wpositive, fatherId=fReference[0]}
  [560] = {x=-187.544, y=-96.686, z=88, rx=-180, rz=61.364, shoulder=lefty, elbow=epositive, wrist=wpositive, fatherId=fReference[0]}
  [561] = {x=-182.731, y=-105.5, z=88, rx=180, rz=58.636, shoulder=lefty, elbow=epositive, wrist=wpositive, fatherId=fReference[0]}
  [562] = {x=-177.505, y=-114.075, z=88, rx=180, rz=55.909, shoulder=lefty, elbow=epositive, wrist=wpositive, fatherId=fReference[0]}
  [563] = {x=-171.876, y=-122.392, z=88, rx=-180, rz=53.182, shoulder=lefty, elbow=epositive, wrist=wpositive, fatherId=fReference[0]}
  [564] = {x=-165.857, y=-130.432, z=88, rx=-180, rz=50.455, shoulder=lefty, elbow=epositive, wrist=wpositive, fatherId=fReference[0]}
  [565] = {x=-159.463, y=-138.176, z=88, rx=-180, rz=47.727, shoulder=lefty, elbow=epositive, wrist=wpositive, fatherId=fReference[0]}
  [566] = {x=-152.708, y=-145.607, z=88, rx=-180, rz=45, shoulder=lefty, elbow=epositive, wrist=wpositive, fatherId=fReference[0]}
  [567] = {x=-145.607, y=-152.708, z=88, rx=-180, rz=42.273, shoulder=lefty, elbow=epositive, wrist=wpositive, fatherId=fReference[0]}
  [568] = {x=-138.176, y=-159.463, z=88, rx=-180, rz=39.545, shoulder=lefty, elbow=epositive, wrist=wpositive, fatherId=fReference[0]}
  [569] = {x=-130.432, y=-165.857, z=88, rx=-180, rz=36.818, shoulder=lefty, elbow=epositive, wrist=wpositive, fatherId=fReference[0]}
  [570] = {x=-122.392, y=-171.876, z=88, rx=-180, rz=34.091, shoulder=lefty, elbow=epositive, wrist=wpositive, fatherId=fReference[0]}
  [571] = {x=-114.075, y=-177.505, z=88, rx=-180, rz=31.364, shoulder=lefty, elbow=epositive, wrist=wpositive, fatherId=fReference[0]}
  [572] = {x=-105.5, y=-182.731, z=88, rx=180, rz=28.636, shoulder=lefty, elbow=epositive, wrist=wpositive, fatherId=fReference[0]}
  [573] = {x=-96.686, y=-187.544, z=88, rx=-180, rz=25.909, shoulder=lefty, elbow=epositive, wrist=wpositive, fatherId=fReference[0]}
  [574] = {x=-87.653, y=-191.932, z=88, rx=-180, rz=23.182, shoulder=lefty, elbow=epositive, wrist=wpositive, fatherId=fReference[0]}
  [575] = {x=-78.421, y=-195.886, z=88, rx=-180, rz=20.455, shoulder=lefty, elbow=epositive, wrist=wpositive, fatherId=fReference[0]}
  [576] = {x=-69.011, y=-199.395, z=88, rx=180, rz=17.727, shoulder=lefty, elbow=epositive, wrist=wpositive, fatherId=fReference[0]}
  [577] = {x=-59.446, y=-202.453, z=88, rx=-180, rz=15, shoulder=lefty, elbow=epositive, wrist=wpositive, fatherId=fReference[0]}
  [578] = {x=-49.745, y=-205.052, z=88, rx=-180, rz=12.273, shoulder=lefty, elbow=epositive, wrist=wpositive, fatherId=fReference[0]}
  [579] = {x=-39.932, y=-207.187, z=88, rx=180, rz=9.545, shoulder=lefty, elbow=epositive, wrist=wpositive, fatherId=fReference[0]}
  [580] = {x=-30.028, y=-208.852, z=88, rx=180, rz=6.818, shoulder=lefty, elbow=epositive, wrist=wpositive, fatherId=fReference[0]}
  [581] = {x=-20.057, y=-210.045, z=88, rx=-180, rz=4.091, shoulder=lefty, elbow=epositive, wrist=wpositive, fatherId=fReference[0]}
  [582] = {x=-10.04, y=-210.761, z=88, rx=-180, rz=1.364, shoulder=lefty, elbow=epositive, wrist=wpositive, fatherId=fReference[0]}
  [583] = {y=-211, z=88, rx=180, rz=-1.364, shoulder=lefty, elbow=epositive, wrist=wpositive, fatherId=fReference[0]}
  [584] = {x=10.04, y=-210.761, z=88, rx=-180, rz=-4.091, shoulder=lefty, elbow=epositive, wrist=wpositive, fatherId=fReference[0]}
  [585] = {x=20.057, y=-210.045, z=88, rx=-180, rz=-6.818, shoulder=lefty, elbow=epositive, wrist=wpositive, fatherId=fReference[0]}
  [586] = {x=30.028, y=-208.852, z=88, rx=-180, rz=-9.545, shoulder=lefty, elbow=epositive, wrist=wpositive, fatherId=fReference[0]}
  [587] = {x=39.932, y=-207.187, z=88, rx=180, rz=-12.273, shoulder=lefty, elbow=epositive, wrist=wpositive, fatherId=fReference[0]}
  [588] = {x=49.745, y=-205.052, z=88, rx=180, rz=-15, shoulder=lefty, elbow=epositive, wrist=wpositive, fatherId=fReference[0]}
  [589] = {x=59.446, y=-202.453, z=88, rx=-180, rz=-17.727, shoulder=lefty, elbow=epositive, wrist=wpositive, fatherId=fReference[0]}
  [590] = {x=69.011, y=-199.395, z=88, rx=180, rz=-20.455, shoulder=lefty, elbow=epositive, wrist=wpositive, fatherId=fReference[0]}
  [591] = {x=78.421, y=-195.886, z=88, rx=-180, rz=-23.182, shoulder=lefty, elbow=epositive, wrist=wpositive, fatherId=fReference[0]}
  [592] = {x=87.653, y=-191.932, z=88, rx=180, rz=-25.909, shoulder=lefty, elbow=epositive, wrist=wpositive, fatherId=fReference[0]}
  [593] = {x=96.686, y=-187.544, z=88, rx=180, rz=-28.636, shoulder=lefty, elbow=epositive, wrist=wpositive, fatherId=fReference[0]}
  [594] = {x=105.5, y=-182.731, z=88, rx=180, rz=-31.364, shoulder=lefty, elbow=epositive, wrist=wpositive, fatherId=fReference[0]}
  [595] = {x=114.075, y=-177.505, z=88, rx=-180, rz=-34.091, shoulder=lefty, elbow=epositive, wrist=wpositive, fatherId=fReference[0]}
  [596] = {x=122.392, y=-171.876, z=88, rx=-180, rz=-36.818, shoulder=lefty, elbow=epositive, wrist=wpositive, fatherId=fReference[0]}
  [597] = {x=130.432, y=-165.857, z=88, rx=180, rz=-39.545, shoulder=lefty, elbow=epositive, wrist=wpositive, fatherId=fReference[0]}
  [598] = {x=138.176, y=-159.463, z=88, rx=180, rz=-42.273, shoulder=lefty, elbow=epositive, wrist=wpositive, fatherId=fReference[0]}
  [599] = {x=145.607, y=-152.708, z=88, rx=180, rz=-45, shoulder=lefty, elbow=epositive, wrist=wpositive, fatherId=fReference[0]}
  [600] = {x=152.708, y=-145.607, z=88, rx=180, rz=-47.727, shoulder=lefty, elbow=epositive, wrist=wpositive, fatherId=fReference[0]}
  [601] = {x=159.463, y=-138.176, z=88, rx=180, rz=-50.455, shoulder=lefty, elbow=epositive, wrist=wpositive, fatherId=fReference[0]}
  [602] = {x=165.857, y=-130.432, z=88, rx=-180, rz=-53.182, shoulder=lefty, elbow=epositive, wrist=wpositive, fatherId=fReference[0]}
  [603] = {x=171.876, y=-122.392, z=88, rx=180, rz=-55.909, shoulder=lefty, elbow=epositive, wrist=wpositive, fatherId=fReference[0]}
  [604] = {x=177.505, y=-114.075, z=88, rx=180, rz=-58.636, shoulder=lefty, elbow=epositive, wrist=wpositive, fatherId=fReference[0]}
  [605] = {x=182.731, y=-105.5, z=88, rx=180, rz=-61.364, shoulder=lefty, elbow=epositive, wrist=wpositive, fatherId=fReference[0]}
  [606] = {x=187.544, y=-96.686, z=88, rx=180, rz=-64.091, shoulder=lefty, elbow=epositive, wrist=wpositive, fatherId=fReference[0]}
  [607] = {x=191.932, y=-87.653, z=88, rx=180, rz=-66.818, shoulder=lefty, elbow=epositive, wrist=wpositive, fatherId=fReference[0]}
  [608] = {x=195.886, y=-78.421, z=88, rx=180, rz=-69.545, shoulder=lefty, elbow=epositive, wrist=wpositive, fatherId=fReference[0]}
  [609] = {x=199.395, y=-69.011, z=88, rx=180, rz=-72.273, shoulder=lefty, elbow=epositive, wrist=wpositive, fatherId=fReference[0]}
  [610] = {x=202.453, y=-59.446, z=88, rx=180, rz=-75, shoulder=lefty, elbow=epositive, wrist=wpositive, fatherId=fReference[0]}
  [611] = {x=205.052, y=-49.745, z=88, rx=180, rz=-77.727, shoulder=lefty, elbow=epositive, wrist=wpositive, fatherId=fReference[0]}
  [612] = {x=207.187, y=-39.932, z=88, rx=180, rz=-80.455, shoulder=lefty, elbow=epositive, wrist=wpositive, fatherId=fReference[0]}
  [613] = {x=208.852, y=-30.028, z=88, rx=180, rz=-83.182, shoulder=lefty, elbow=epositive, wrist=wpositive, fatherId=fReference[0]}
  [614] = {x=210.045, y=-20.057, z=88, rx=180, rz=-85.909, shoulder=lefty, elbow=epositive, wrist=wpositive, fatherId=fReference[0]}
  [615] = {x=210.761, y=-10.04, z=88, rx=180, rz=-88.636, shoulder=lefty, elbow=epositive, wrist=wpositive, fatherId=fReference[0]}
  [616] = {x=211, z=88, rx=-180, rz=-91.364, shoulder=lefty, elbow=epositive, wrist=wpositive, fatherId=fReference[0]}
  [617] = {x=210.761, y=10.04, z=88, rx=-180, rz=-94.091, shoulder=lefty, elbow=epositive, wrist=wpositive, fatherId=fReference[0]}
  [618] = {x=210.045, y=20.057, z=88, rx=-180, rz=-96.818, shoulder=lefty, elbow=epositive, wrist=wpositive, fatherId=fReference[0]}
  [619] = {x=208.852, y=30.028, z=88, rx=-180, rz=-99.545, shoulder=lefty, elbow=epositive, wrist=wpositive, fatherId=fReference[0]}
  [620] = {x=207.187, y=39.932, z=88, rx=-180, rz=-102.273, shoulder=lefty, elbow=epositive, wrist=wpositive, fatherId=fReference[0]}
  [621] = {x=205.052, y=49.745, z=88, rx=-180, rz=-105, shoulder=lefty, elbow=epositive, wrist=wpositive, fatherId=fReference[0]}
  [622] = {x=202.453, y=59.446, z=88, rx=-180, rz=-107.727, shoulder=lefty, elbow=epositive, wrist=wpositive, fatherId=fReference[0]}
  [623] = {x=199.395, y=69.011, z=88, rx=-180, rz=-110.455, shoulder=lefty, elbow=epositive, wrist=wpositive, fatherId=fReference[0]}
  [624] = {x=195.886, y=78.421, z=88, rx=-180, rz=-113.182, shoulder=lefty, elbow=epositive, wrist=wpositive, fatherId=fReference[0]}
  [625] = {x=191.932, y=87.653, z=88, rx=-180, rz=-115.909, shoulder=lefty, elbow=epositive, wrist=wpositive, fatherId=fReference[0]}
  [626] = {x=187.544, y=96.686, z=88, rx=-180, rz=-118.636, shoulder=lefty, elbow=epositive, wrist=wpositive, fatherId=fReference[0]}
  [627] = {x=182.731, y=105.5, z=88, rx=-180, rz=-121.364, shoulder=lefty, elbow=epositive, wrist=wpositive, fatherId=fReference[0]}
  [628] = {x=177.505, y=114.075, z=88, rx=-180, rz=-124.091, shoulder=lefty, elbow=epositive, wrist=wpositive, fatherId=fReference[0]}
  [629] = {x=171.876, y=122.392, z=88, rx=-180, rz=-126.818, shoulder=lefty, elbow=epositive, wrist=wpositive, fatherId=fReference[0]}
  [630] = {x=165.857, y=130.432, z=88, rx=180, rz=-129.545, shoulder=lefty, elbow=epositive, wrist=wpositive, fatherId=fReference[0]}
  [631] = {x=159.463, y=138.176, z=88, rx=-180, rz=-132.273, shoulder=lefty, elbow=epositive, wrist=wpositive, fatherId=fReference[0]}
  [632] = {x=152.708, y=145.607, z=88, rx=-180, rz=-135, shoulder=lefty, elbow=epositive, wrist=wpositive, fatherId=fReference[0]}
  [633] = {x=145.607, y=152.708, z=88, rx=-180, rz=-137.727, shoulder=lefty, elbow=epositive, wrist=wpositive, fatherId=fReference[0]}
  [634] = {x=138.176, y=159.463, z=88, rx=-180, rz=-140.455, shoulder=lefty, elbow=epositive, wrist=wpositive, fatherId=fReference[0]}
  [635] = {x=130.432, y=165.857, z=88, rx=-180, rz=-143.182, shoulder=lefty, elbow=epositive, wrist=wpositive, fatherId=fReference[0]}
  [636] = {x=122.392, y=171.876, z=88, rx=-180, rz=-145.909, shoulder=lefty, elbow=epositive, wrist=wpositive, fatherId=fReference[0]}
  [637] = {x=114.075, y=177.505, z=88, rx=-180, rz=-148.636, shoulder=lefty, elbow=epositive, wrist=wpositive, fatherId=fReference[0]}
  [638] = {x=105.5, y=182.731, z=88, rx=-180, rz=-151.364, shoulder=lefty, elbow=epositive, wrist=wpositive, fatherId=fReference[0]}
  [639] = {x=96.686, y=187.544, z=88, rx=-180, rz=-154.091, shoulder=lefty, elbow=epositive, wrist=wpositive, fatherId=fReference[0]}
  [640] = {x=87.653, y=191.932, z=88, rx=-180, rz=-156.818, shoulder=lefty, elbow=epositive, wrist=wpositive, fatherId=fReference[0]}
  [641] = {x=78.421, y=195.886, z=88, rx=-180, rz=-159.545, shoulder=lefty, elbow=epositive, wrist=wpositive, fatherId=fReference[0]}
  [642] = {x=69.011, y=199.395, z=88, rx=-180, rz=-162.273, shoulder=lefty, elbow=epositive, wrist=wpositive, fatherId=fReference[0]}
  [643] = {x=59.446, y=202.453, z=88, rx=-180, rz=-165, shoulder=lefty, elbow=epositive, wrist=wpositive, fatherId=fReference[0]}
  [644] = {x=49.745, y=205.052, z=88, rx=180, rz=-167.727, shoulder=lefty, elbow=epositive, wrist=wpositive, fatherId=fReference[0]}
  [645] = {x=39.932, y=207.187, z=88, rx=-180, rz=-170.455, shoulder=lefty, elbow=epositive, wrist=wpositive, fatherId=fReference[0]}
  [646] = {x=30.028, y=208.852, z=88, rx=-180, rz=-173.182, shoulder=lefty, elbow=epositive, wrist=wpositive, fatherId=fReference[0]}
  [647] = {x=20.057, y=210.045, z=88, rx=-180, rz=-175.909, shoulder=lefty, elbow=epositive, wrist=wpositive, fatherId=fReference[0]}
  [648] = {x=10.04, y=210.761, z=88, rx=180, rz=-178.636, shoulder=lefty, elbow=epositive, wrist=wpositive, fatherId=fReference[0]}
  [649] = {y=211, z=88, rx=180, rz=178.636, shoulder=lefty, elbow=epositive, wrist=wpositive, fatherId=fReference[0]}
  [650] = {x=-10.04, y=210.761, z=88, rx=-180, rz=175.909, shoulder=lefty, elbow=epositive, wrist=wpositive, fatherId=fReference[0]}
  [651] = {x=-20.057, y=210.045, z=88, rx=-180, rz=173.182, shoulder=lefty, elbow=epositive, wrist=wpositive, fatherId=fReference[0]}
  [652] = {x=-30.028, y=208.852, z=88, rx=-180, rz=170.455, shoulder=lefty, elbow=epositive, wrist=wpositive, fatherId=fReference[0]}
  [653] = {x=-39.932, y=207.187, z=88, rx=180, rz=167.727, shoulder=lefty, elbow=epositive, wrist=wpositive, fatherId=fReference[0]}
  [654] = {x=-49.745, y=205.052, z=88, rx=-180, rz=165, shoulder=lefty, elbow=epositive, wrist=wpositive, fatherId=fReference[0]}
  [655] = {x=-59.446, y=202.453, z=88, rx=-180, rz=162.273, shoulder=lefty, elbow=epositive, wrist=wpositive, fatherId=fReference[0]}
  [656] = {x=-69.011, y=199.395, z=88, rx=180, rz=159.545, shoulder=lefty, elbow=epositive, wrist=wpositive, fatherId=fReference[0]}
  [657] = {x=-78.421, y=195.886, z=88, rx=180, rz=156.818, shoulder=lefty, elbow=epositive, wrist=wpositive, fatherId=fReference[0]}
  [658] = {x=-87.653, y=191.932, z=88, rx=-180, rz=154.091, shoulder=lefty, elbow=epositive, wrist=wpositive, fatherId=fReference[0]}
  [659] = {x=-96.686, y=187.544, z=88, rx=-180, rz=151.364, shoulder=lefty, elbow=epositive, wrist=wpositive, fatherId=fReference[0]}
  [660] = {x=-105.5, y=182.731, z=88, rx=180, rz=148.636, shoulder=lefty, elbow=epositive, wrist=wpositive, fatherId=fReference[0]}
  [661] = {x=-114.075, y=177.505, z=88, rx=180, rz=145.909, shoulder=lefty, elbow=epositive, wrist=wpositive, fatherId=fReference[0]}
  [662] = {x=-122.392, y=171.876, z=88, rx=-180, rz=143.182, shoulder=lefty, elbow=epositive, wrist=wpositive, fatherId=fReference[0]}
  [663] = {x=-130.432, y=165.857, z=88, rx=180, rz=140.455, shoulder=lefty, elbow=epositive, wrist=wpositive, fatherId=fReference[0]}
  [664] = {x=-138.176, y=159.463, z=88, rx=180, rz=137.727, shoulder=lefty, elbow=epositive, wrist=wpositive, fatherId=fReference[0]}
  [665] = {x=-145.607, y=152.708, z=88, rx=-180, rz=135, shoulder=lefty, elbow=epositive, wrist=wpositive, fatherId=fReference[0]}
  [666] = {x=-152.708, y=145.607, z=88, rx=180, rz=132.273, shoulder=lefty, elbow=epositive, wrist=wpositive, fatherId=fReference[0]}
  [667] = {x=-159.463, y=138.176, z=88, rx=180, rz=129.545, shoulder=lefty, elbow=epositive, wrist=wpositive, fatherId=fReference[0]}
  [668] = {x=-165.857, y=130.432, z=88, rx=180, rz=126.818, shoulder=lefty, elbow=epositive, wrist=wpositive, fatherId=fReference[0]}
  [669] = {x=-171.876, y=122.392, z=88, rx=180, rz=124.091, shoulder=lefty, elbow=epositive, wrist=wpositive, fatherId=fReference[0]}
  [670] = {x=-177.505, y=114.075, z=88, rx=180, rz=121.364, shoulder=lefty, elbow=epositive, wrist=wpositive, fatherId=fReference[0]}
  [671] = {x=-182.731, y=105.5, z=88, rx=180, rz=118.636, shoulder=lefty, elbow=epositive, wrist=wpositive, fatherId=fReference[0]}
  [672] = {x=-187.544, y=96.686, z=88, rx=180, rz=115.909, shoulder=lefty, elbow=epositive, wrist=wpositive, fatherId=fReference[0]}
  [673] = {x=-191.932, y=87.653, z=88, rx=180, rz=113.182, shoulder=lefty, elbow=epositive, wrist=wpositive, fatherId=fReference[0]}
  [674] = {x=-195.886, y=78.421, z=88, rx=-180, rz=110.455, shoulder=lefty, elbow=epositive, wrist=wpositive, fatherId=fReference[0]}
  [675] = {x=-199.395, y=69.011, z=88, rx=180, rz=107.727, shoulder=lefty, elbow=epositive, wrist=wpositive, fatherId=fReference[0]}
  [676] = {x=-202.453, y=59.446, z=88, rx=180, rz=105, shoulder=lefty, elbow=epositive, wrist=wpositive, fatherId=fReference[0]}
  [677] = {x=-205.052, y=49.745, z=88, rx=180, rz=102.273, shoulder=lefty, elbow=epositive, wrist=wpositive, fatherId=fReference[0]}
  [678] = {x=-207.187, y=39.932, z=88, rx=180, rz=99.545, shoulder=lefty, elbow=epositive, wrist=wpositive, fatherId=fReference[0]}
  [679] = {x=-208.852, y=30.028, z=88, rx=180, rz=96.818, shoulder=lefty, elbow=epositive, wrist=wpositive, fatherId=fReference[0]}
  [680] = {x=-210.045, y=20.057, z=88, rx=180, rz=94.091, shoulder=lefty, elbow=epositive, wrist=wpositive, fatherId=fReference[0]}
  [681] = {x=-210.761, y=10.04, z=88, rx=180, rz=91.364, shoulder=lefty, elbow=epositive, wrist=wpositive, fatherId=fReference[0]}
  [682] = {x=-211, z=88, rx=180, rz=91.364, shoulder=lefty, elbow=epositive, wrist=wpositive, fatherId=fReference[0]}
  [683] = {x=-211, z=88, rx=180, rz=91.364, shoulder=lefty, elbow=epositive, wrist=wpositive, fatherId=fReference[0]}
  [684] = {x=-211, z=188, rx=180, rz=91.364, shoulder=lefty, elbow=epositive, wrist=wpositive, fatherId=fReference[0]}
  [685] = {x=-211, z=210, rx=180, rz=91.364, shoulder=lefty, elbow=epositive, wrist=wpositive, fatherId=fReference[0]}
  [686] = {x=-211, z=110, rx=180, rz=91.364, shoulder=lefty, elbow=epositive, wrist=wpositive, fatherId=fReference[0]}
  [687] = {x=-211, z=110, rx=180, rz=91.364, shoulder=lefty, elbow=epositive, wrist=wpositive, fatherId=fReference[0]}
  [688] = {x=-210.761, y=10.04, z=110, rx=180, rz=94.091, shoulder=lefty, elbow=epositive, wrist=wpositive, fatherId=fReference[0]}
  [689] = {x=-210.045, y=20.057, z=110, rx=180, rz=96.818, shoulder=lefty, elbow=epositive, wrist=wpositive, fatherId=fReference[0]}
  [690] = {x=-208.852, y=30.028, z=110, rx=180, rz=99.545, shoulder=lefty, elbow=epositive, wrist=wpositive, fatherId=fReference[0]}
  [691] = {x=-207.187, y=39.932, z=110, rx=180, rz=102.273, shoulder=lefty, elbow=epositive, wrist=wpositive, fatherId=fReference[0]}
  [692] = {x=-205.052, y=49.745, z=110, rx=180, rz=105, shoulder=lefty, elbow=epositive, wrist=wpositive, fatherId=fReference[0]}
  [693] = {x=-202.453, y=59.446, z=110, rx=180, rz=107.727, shoulder=lefty, elbow=epositive, wrist=wpositive, fatherId=fReference[0]}
  [694] = {x=-199.395, y=69.011, z=110, rx=180, rz=110.455, shoulder=lefty, elbow=epositive, wrist=wpositive, fatherId=fReference[0]}
  [695] = {x=-195.886, y=78.421, z=110, rx=180, rz=113.182, shoulder=lefty, elbow=epositive, wrist=wpositive, fatherId=fReference[0]}
  [696] = {x=-191.932, y=87.653, z=110, rx=180, rz=115.909, shoulder=lefty, elbow=epositive, wrist=wpositive, fatherId=fReference[0]}
  [697] = {x=-187.544, y=96.686, z=110, rx=180, rz=118.636, shoulder=lefty, elbow=epositive, wrist=wpositive, fatherId=fReference[0]}
  [698] = {x=-182.731, y=105.5, z=110, rx=180, rz=121.364, shoulder=lefty, elbow=epositive, wrist=wpositive, fatherId=fReference[0]}
  [699] = {x=-177.505, y=114.075, z=110, rx=180, rz=124.091, shoulder=lefty, elbow=epositive, wrist=wpositive, fatherId=fReference[0]}
  [700] = {x=-171.876, y=122.392, z=110, rx=180, rz=126.818, shoulder=lefty, elbow=epositive, wrist=wpositive, fatherId=fReference[0]}
  [701] = {x=-165.857, y=130.432, z=110, rx=180, rz=129.545, shoulder=lefty, elbow=epositive, wrist=wpositive, fatherId=fReference[0]}
  [702] = {x=-159.463, y=138.176, z=110, rx=180, rz=132.273, shoulder=lefty, elbow=epositive, wrist=wpositive, fatherId=fReference[0]}
  [703] = {x=-152.708, y=145.607, z=110, rx=-180, rz=135, shoulder=lefty, elbow=epositive, wrist=wpositive, fatherId=fReference[0]}
  [704] = {x=-145.607, y=152.708, z=110, rx=180, rz=137.727, shoulder=lefty, elbow=epositive, wrist=wpositive, fatherId=fReference[0]}
  [705] = {x=-138.176, y=159.463, z=110, rx=180, rz=140.455, shoulder=lefty, elbow=epositive, wrist=wpositive, fatherId=fReference[0]}
  [706] = {x=-130.432, y=165.857, z=110, rx=180, rz=143.182, shoulder=lefty, elbow=epositive, wrist=wpositive, fatherId=fReference[0]}
  [707] = {x=-122.392, y=171.876, z=110, rx=180, rz=145.909, shoulder=lefty, elbow=epositive, wrist=wpositive, fatherId=fReference[0]}
  [708] = {x=-114.075, y=177.505, z=110, rx=-180, rz=148.636, shoulder=lefty, elbow=epositive, wrist=wpositive, fatherId=fReference[0]}
  [709] = {x=-105.5, y=182.731, z=110, rx=180, rz=151.364, shoulder=lefty, elbow=epositive, wrist=wpositive, fatherId=fReference[0]}
  [710] = {x=-96.686, y=187.544, z=110, rx=180, rz=154.091, shoulder=lefty, elbow=epositive, wrist=wpositive, fatherId=fReference[0]}
  [711] = {x=-87.653, y=191.932, z=110, rx=180, rz=156.818, shoulder=lefty, elbow=epositive, wrist=wpositive, fatherId=fReference[0]}
  [712] = {x=-78.421, y=195.886, z=110, rx=-180, rz=159.545, shoulder=lefty, elbow=epositive, wrist=wpositive, fatherId=fReference[0]}
  [713] = {x=-69.011, y=199.395, z=110, rx=180, rz=162.273, shoulder=lefty, elbow=epositive, wrist=wpositive, fatherId=fReference[0]}
  [714] = {x=-59.446, y=202.453, z=110, rx=-180, rz=165, shoulder=lefty, elbow=epositive, wrist=wpositive, fatherId=fReference[0]}
  [715] = {x=-49.745, y=205.052, z=110, rx=180, rz=167.727, shoulder=lefty, elbow=epositive, wrist=wpositive, fatherId=fReference[0]}
  [716] = {x=-39.932, y=207.187, z=110, rx=180, rz=170.455, shoulder=lefty, elbow=epositive, wrist=wpositive, fatherId=fReference[0]}
  [717] = {x=-30.028, y=208.852, z=110, rx=-180, rz=173.182, shoulder=lefty, elbow=epositive, wrist=wpositive, fatherId=fReference[0]}
  [718] = {x=-20.057, y=210.045, z=110, rx=-180, rz=175.909, shoulder=lefty, elbow=epositive, wrist=wpositive, fatherId=fReference[0]}
  [719] = {x=-10.04, y=210.761, z=110, rx=180, rz=178.636, shoulder=lefty, elbow=epositive, wrist=wpositive, fatherId=fReference[0]}
  [720] = {y=211, z=110, rx=180, rz=-178.636, shoulder=lefty, elbow=epositive, wrist=wpositive, fatherId=fReference[0]}
  [721] = {x=10.04, y=210.761, z=110, rx=-180, rz=-175.909, shoulder=lefty, elbow=epositive, wrist=wpositive, fatherId=fReference[0]}
  [722] = {x=20.057, y=210.045, z=110, rx=180, rz=-173.182, shoulder=lefty, elbow=epositive, wrist=wpositive, fatherId=fReference[0]}
  [723] = {x=30.028, y=208.852, z=110, rx=-180, rz=-170.455, shoulder=lefty, elbow=epositive, wrist=wpositive, fatherId=fReference[0]}
  [724] = {x=39.932, y=207.187, z=110, rx=-180, rz=-167.727, shoulder=lefty, elbow=epositive, wrist=wpositive, fatherId=fReference[0]}
  [725] = {x=49.745, y=205.052, z=110, rx=-180, rz=-165, shoulder=lefty, elbow=epositive, wrist=wpositive, fatherId=fReference[0]}
  [726] = {x=59.446, y=202.453, z=110, rx=-180, rz=-162.273, shoulder=lefty, elbow=epositive, wrist=wpositive, fatherId=fReference[0]}
  [727] = {x=69.011, y=199.395, z=110, rx=180, rz=-159.545, shoulder=lefty, elbow=epositive, wrist=wpositive, fatherId=fReference[0]}
  [728] = {x=78.421, y=195.886, z=110, rx=180, rz=-156.818, shoulder=lefty, elbow=epositive, wrist=wpositive, fatherId=fReference[0]}
  [729] = {x=87.653, y=191.932, z=110, rx=-180, rz=-154.091, shoulder=lefty, elbow=epositive, wrist=wpositive, fatherId=fReference[0]}
  [730] = {x=96.686, y=187.544, z=110, rx=180, rz=-151.364, shoulder=lefty, elbow=epositive, wrist=wpositive, fatherId=fReference[0]}
  [731] = {x=105.5, y=182.731, z=110, rx=-180, rz=-148.636, shoulder=lefty, elbow=epositive, wrist=wpositive, fatherId=fReference[0]}
  [732] = {x=114.075, y=177.505, z=110, rx=-180, rz=-145.909, shoulder=lefty, elbow=epositive, wrist=wpositive, fatherId=fReference[0]}
  [733] = {x=122.392, y=171.876, z=110, rx=-180, rz=-143.182, shoulder=lefty, elbow=epositive, wrist=wpositive, fatherId=fReference[0]}
  [734] = {x=130.432, y=165.857, z=110, rx=-180, rz=-140.455, shoulder=lefty, elbow=epositive, wrist=wpositive, fatherId=fReference[0]}
  [735] = {x=138.176, y=159.463, z=110, rx=-180, rz=-137.727, shoulder=lefty, elbow=epositive, wrist=wpositive, fatherId=fReference[0]}
  [736] = {x=145.607, y=152.708, z=110, rx=-180, rz=-135, shoulder=lefty, elbow=epositive, wrist=wpositive, fatherId=fReference[0]}
  [737] = {x=152.708, y=145.607, z=110, rx=-180, rz=-132.273, shoulder=lefty, elbow=epositive, wrist=wpositive, fatherId=fReference[0]}
  [738] = {x=159.463, y=138.176, z=110, rx=-180, rz=-129.545, shoulder=lefty, elbow=epositive, wrist=wpositive, fatherId=fReference[0]}
  [739] = {x=165.857, y=130.432, z=110, rx=-180, rz=-126.818, shoulder=lefty, elbow=epositive, wrist=wpositive, fatherId=fReference[0]}
  [740] = {x=171.876, y=122.392, z=110, rx=-180, rz=-124.091, shoulder=lefty, elbow=epositive, wrist=wpositive, fatherId=fReference[0]}
  [741] = {x=177.505, y=114.075, z=110, rx=-180, rz=-121.364, shoulder=lefty, elbow=epositive, wrist=wpositive, fatherId=fReference[0]}
